(* Logix 5000 project; controller Universal_Device_Info_AOI_V0_1 vendor 1 type 14 code 176 rev 32.11; software revision 32.00; part 4 of 11 *)

           TBEN_L4_8IOL:O.Data[121].5   // IO-Link Port 8 - Output data word 7 (INT bit5)
           TBEN_L4_8IOL:O.Data[121].6   // IO-Link Port 8 - Output data word 7 (INT bit6)
           TBEN_L4_8IOL:O.Data[121].7   // IO-Link Port 8 - Output data word 7 (INT bit7)
           TBEN_L4_8IOL:O.Data[121].8   // IO-Link Port 8 - Output data word 7 (INT bit8)
           TBEN_L4_8IOL:O.Data[121].9   // IO-Link Port 8 - Output data word 7 (INT bit9)
           TBEN_L4_8IOL:O.Data[122]   // IO-Link Port 8 - Output data word 8
           TBEN_L4_8IOL:O.Data[122].0   // IO-Link Port 8 - Output data word 8 (INT bit0)
           TBEN_L4_8IOL:O.Data[122].1   // IO-Link Port 8 - Output data word 8 (INT bit1)
           TBEN_L4_8IOL:O.Data[122].10   // IO-Link Port 8 - Output data word 8 (INT bit10)
           TBEN_L4_8IOL:O.Data[122].11   // IO-Link Port 8 - Output data word 8 (INT bit11)
           TBEN_L4_8IOL:O.Data[122].12   // IO-Link Port 8 - Output data word 8 (INT bit12)
           TBEN_L4_8IOL:O.Data[122].13   // IO-Link Port 8 - Output data word 8 (INT bit13)
           TBEN_L4_8IOL:O.Data[122].14   // IO-Link Port 8 - Output data word 8 (INT bit14)
           TBEN_L4_8IOL:O.Data[122].15   // IO-Link Port 8 - Output data word 8 (INT bit15)
           TBEN_L4_8IOL:O.Data[122].2   // IO-Link Port 8 - Output data word 8 (INT bit2)
           TBEN_L4_8IOL:O.Data[122].3   // IO-Link Port 8 - Output data word 8 (INT bit3)
           TBEN_L4_8IOL:O.Data[122].4   // IO-Link Port 8 - Output data word 8 (INT bit4)
           TBEN_L4_8IOL:O.Data[122].5   // IO-Link Port 8 - Output data word 8 (INT bit5)
           TBEN_L4_8IOL:O.Data[122].6   // IO-Link Port 8 - Output data word 8 (INT bit6)
           TBEN_L4_8IOL:O.Data[122].7   // IO-Link Port 8 - Output data word 8 (INT bit7)
           TBEN_L4_8IOL:O.Data[122].8   // IO-Link Port 8 - Output data word 8 (INT bit8)
           TBEN_L4_8IOL:O.Data[122].9   // IO-Link Port 8 - Output data word 8 (INT bit9)
           TBEN_L4_8IOL:O.Data[123]   // IO-Link Port 8 - Output data word 9
           TBEN_L4_8IOL:O.Data[123].0   // IO-Link Port 8 - Output data word 9 (INT bit0)
           TBEN_L4_8IOL:O.Data[123].1   // IO-Link Port 8 - Output data word 9 (INT bit1)
           TBEN_L4_8IOL:O.Data[123].10   // IO-Link Port 8 - Output data word 9 (INT bit10)
           TBEN_L4_8IOL:O.Data[123].11   // IO-Link Port 8 - Output data word 9 (INT bit11)
           TBEN_L4_8IOL:O.Data[123].12   // IO-Link Port 8 - Output data word 9 (INT bit12)
           TBEN_L4_8IOL:O.Data[123].13   // IO-Link Port 8 - Output data word 9 (INT bit13)
           TBEN_L4_8IOL:O.Data[123].14   // IO-Link Port 8 - Output data word 9 (INT bit14)
           TBEN_L4_8IOL:O.Data[123].15   // IO-Link Port 8 - Output data word 9 (INT bit15)
           TBEN_L4_8IOL:O.Data[123].2   // IO-Link Port 8 - Output data word 9 (INT bit2)
           TBEN_L4_8IOL:O.Data[123].3   // IO-Link Port 8 - Output data word 9 (INT bit3)
           TBEN_L4_8IOL:O.Data[123].4   // IO-Link Port 8 - Output data word 9 (INT bit4)
           TBEN_L4_8IOL:O.Data[123].5   // IO-Link Port 8 - Output data word 9 (INT bit5)
           TBEN_L4_8IOL:O.Data[123].6   // IO-Link Port 8 - Output data word 9 (INT bit6)
           TBEN_L4_8IOL:O.Data[123].7   // IO-Link Port 8 - Output data word 9 (INT bit7)
           TBEN_L4_8IOL:O.Data[123].8   // IO-Link Port 8 - Output data word 9 (INT bit8)
           TBEN_L4_8IOL:O.Data[123].9   // IO-Link Port 8 - Output data word 9 (INT bit9)
           TBEN_L4_8IOL:O.Data[124]   // IO-Link Port 8 - Output data word 10
           TBEN_L4_8IOL:O.Data[124].0   // IO-Link Port 8 - Output data word 10 (INT bit0)
           TBEN_L4_8IOL:O.Data[124].1   // IO-Link Port 8 - Output data word 10 (INT bit1)
           TBEN_L4_8IOL:O.Data[124].10   // IO-Link Port 8 - Output data word 10 (INT bit10)
           TBEN_L4_8IOL:O.Data[124].11   // IO-Link Port 8 - Output data word 10 (INT bit11)
           TBEN_L4_8IOL:O.Data[124].12   // IO-Link Port 8 - Output data word 10 (INT bit12)
           TBEN_L4_8IOL:O.Data[124].13   // IO-Link Port 8 - Output data word 10 (INT bit13)
           TBEN_L4_8IOL:O.Data[124].14   // IO-Link Port 8 - Output data word 10 (INT bit14)
           TBEN_L4_8IOL:O.Data[124].15   // IO-Link Port 8 - Output data word 10 (INT bit15)
           TBEN_L4_8IOL:O.Data[124].2   // IO-Link Port 8 - Output data word 10 (INT bit2)
           TBEN_L4_8IOL:O.Data[124].3   // IO-Link Port 8 - Output data word 10 (INT bit3)
           TBEN_L4_8IOL:O.Data[124].4   // IO-Link Port 8 - Output data word 10 (INT bit4)
           TBEN_L4_8IOL:O.Data[124].5   // IO-Link Port 8 - Output data word 10 (INT bit5)
           TBEN_L4_8IOL:O.Data[124].6   // IO-Link Port 8 - Output data word 10 (INT bit6)
           TBEN_L4_8IOL:O.Data[124].7   // IO-Link Port 8 - Output data word 10 (INT bit7)
           TBEN_L4_8IOL:O.Data[124].8   // IO-Link Port 8 - Output data word 10 (INT bit8)
           TBEN_L4_8IOL:O.Data[124].9   // IO-Link Port 8 - Output data word 10 (INT bit9)
           TBEN_L4_8IOL:O.Data[125]   // IO-Link Port 8 - Output data word 11
           TBEN_L4_8IOL:O.Data[125].0   // IO-Link Port 8 - Output data word 11 (INT bit0)
           TBEN_L4_8IOL:O.Data[125].1   // IO-Link Port 8 - Output data word 11 (INT bit1)
           TBEN_L4_8IOL:O.Data[125].10   // IO-Link Port 8 - Output data word 11 (INT bit10)
           TBEN_L4_8IOL:O.Data[125].11   // IO-Link Port 8 - Output data word 11 (INT bit11)
           TBEN_L4_8IOL:O.Data[125].12   // IO-Link Port 8 - Output data word 11 (INT bit12)
           TBEN_L4_8IOL:O.Data[125].13   // IO-Link Port 8 - Output data word 11 (INT bit13)
           TBEN_L4_8IOL:O.Data[125].14   // IO-Link Port 8 - Output data word 11 (INT bit14)
           TBEN_L4_8IOL:O.Data[125].15   // IO-Link Port 8 - Output data word 11 (INT bit15)
           TBEN_L4_8IOL:O.Data[125].2   // IO-Link Port 8 - Output data word 11 (INT bit2)
           TBEN_L4_8IOL:O.Data[125].3   // IO-Link Port 8 - Output data word 11 (INT bit3)
           TBEN_L4_8IOL:O.Data[125].4   // IO-Link Port 8 - Output data word 11 (INT bit4)
           TBEN_L4_8IOL:O.Data[125].5   // IO-Link Port 8 - Output data word 11 (INT bit5)
           TBEN_L4_8IOL:O.Data[125].6   // IO-Link Port 8 - Output data word 11 (INT bit6)
           TBEN_L4_8IOL:O.Data[125].7   // IO-Link Port 8 - Output data word 11 (INT bit7)
           TBEN_L4_8IOL:O.Data[125].8   // IO-Link Port 8 - Output data word 11 (INT bit8)
           TBEN_L4_8IOL:O.Data[125].9   // IO-Link Port 8 - Output data word 11 (INT bit9)
           TBEN_L4_8IOL:O.Data[126]   // IO-Link Port 8 - Output data word 12
           TBEN_L4_8IOL:O.Data[126].0   // IO-Link Port 8 - Output data word 12 (INT bit0)
           TBEN_L4_8IOL:O.Data[126].1   // IO-Link Port 8 - Output data word 12 (INT bit1)
           TBEN_L4_8IOL:O.Data[126].10   // IO-Link Port 8 - Output data word 12 (INT bit10)
           TBEN_L4_8IOL:O.Data[126].11   // IO-Link Port 8 - Output data word 12 (INT bit11)
           TBEN_L4_8IOL:O.Data[126].12   // IO-Link Port 8 - Output data word 12 (INT bit12)
           TBEN_L4_8IOL:O.Data[126].13   // IO-Link Port 8 - Output data word 12 (INT bit13)
           TBEN_L4_8IOL:O.Data[126].14   // IO-Link Port 8 - Output data word 12 (INT bit14)
           TBEN_L4_8IOL:O.Data[126].15   // IO-Link Port 8 - Output data word 12 (INT bit15)
           TBEN_L4_8IOL:O.Data[126].2   // IO-Link Port 8 - Output data word 12 (INT bit2)
           TBEN_L4_8IOL:O.Data[126].3   // IO-Link Port 8 - Output data word 12 (INT bit3)
           TBEN_L4_8IOL:O.Data[126].4   // IO-Link Port 8 - Output data word 12 (INT bit4)
           TBEN_L4_8IOL:O.Data[126].5   // IO-Link Port 8 - Output data word 12 (INT bit5)
           TBEN_L4_8IOL:O.Data[126].6   // IO-Link Port 8 - Output data word 12 (INT bit6)
           TBEN_L4_8IOL:O.Data[126].7   // IO-Link Port 8 - Output data word 12 (INT bit7)
           TBEN_L4_8IOL:O.Data[126].8   // IO-Link Port 8 - Output data word 12 (INT bit8)
           TBEN_L4_8IOL:O.Data[126].9   // IO-Link Port 8 - Output data word 12 (INT bit9)
           TBEN_L4_8IOL:O.Data[127]   // IO-Link Port 8 - Output data word 13
           TBEN_L4_8IOL:O.Data[127].0   // IO-Link Port 8 - Output data word 13 (INT bit0)
           TBEN_L4_8IOL:O.Data[127].1   // IO-Link Port 8 - Output data word 13 (INT bit1)
           TBEN_L4_8IOL:O.Data[127].10   // IO-Link Port 8 - Output data word 13 (INT bit10)
           TBEN_L4_8IOL:O.Data[127].11   // IO-Link Port 8 - Output data word 13 (INT bit11)
           TBEN_L4_8IOL:O.Data[127].12   // IO-Link Port 8 - Output data word 13 (INT bit12)
           TBEN_L4_8IOL:O.Data[127].13   // IO-Link Port 8 - Output data word 13 (INT bit13)
           TBEN_L4_8IOL:O.Data[127].14   // IO-Link Port 8 - Output data word 13 (INT bit14)
           TBEN_L4_8IOL:O.Data[127].15   // IO-Link Port 8 - Output data word 13 (INT bit15)
           TBEN_L4_8IOL:O.Data[127].2   // IO-Link Port 8 - Output data word 13 (INT bit2)
           TBEN_L4_8IOL:O.Data[127].3   // IO-Link Port 8 - Output data word 13 (INT bit3)
           TBEN_L4_8IOL:O.Data[127].4   // IO-Link Port 8 - Output data word 13 (INT bit4)
           TBEN_L4_8IOL:O.Data[127].5   // IO-Link Port 8 - Output data word 13 (INT bit5)
           TBEN_L4_8IOL:O.Data[127].6   // IO-Link Port 8 - Output data word 13 (INT bit6)
           TBEN_L4_8IOL:O.Data[127].7   // IO-Link Port 8 - Output data word 13 (INT bit7)
           TBEN_L4_8IOL:O.Data[127].8   // IO-Link Port 8 - Output data word 13 (INT bit8)
           TBEN_L4_8IOL:O.Data[127].9   // IO-Link Port 8 - Output data word 13 (INT bit9)
           TBEN_L4_8IOL:O.Data[128]   // IO-Link Port 8 - Output data word 14
           TBEN_L4_8IOL:O.Data[128].0   // IO-Link Port 8 - Output data word 14 (INT bit0)
           TBEN_L4_8IOL:O.Data[128].1   // IO-Link Port 8 - Output data word 14 (INT bit1)
           TBEN_L4_8IOL:O.Data[128].10   // IO-Link Port 8 - Output data word 14 (INT bit10)
           TBEN_L4_8IOL:O.Data[128].11   // IO-Link Port 8 - Output data word 14 (INT bit11)
           TBEN_L4_8IOL:O.Data[128].12   // IO-Link Port 8 - Output data word 14 (INT bit12)
           TBEN_L4_8IOL:O.Data[128].13   // IO-Link Port 8 - Output data word 14 (INT bit13)
           TBEN_L4_8IOL:O.Data[128].14   // IO-Link Port 8 - Output data word 14 (INT bit14)
           TBEN_L4_8IOL:O.Data[128].15   // IO-Link Port 8 - Output data word 14 (INT bit15)
           TBEN_L4_8IOL:O.Data[128].2   // IO-Link Port 8 - Output data word 14 (INT bit2)
           TBEN_L4_8IOL:O.Data[128].3   // IO-Link Port 8 - Output data word 14 (INT bit3)
           TBEN_L4_8IOL:O.Data[128].4   // IO-Link Port 8 - Output data word 14 (INT bit4)
           TBEN_L4_8IOL:O.Data[128].5   // IO-Link Port 8 - Output data word 14 (INT bit5)
           TBEN_L4_8IOL:O.Data[128].6   // IO-Link Port 8 - Output data word 14 (INT bit6)
           TBEN_L4_8IOL:O.Data[128].7   // IO-Link Port 8 - Output data word 14 (INT bit7)
           TBEN_L4_8IOL:O.Data[128].8   // IO-Link Port 8 - Output data word 14 (INT bit8)
           TBEN_L4_8IOL:O.Data[128].9   // IO-Link Port 8 - Output data word 14 (INT bit9)
           TBEN_L4_8IOL:O.Data[129]   // IO-Link Port 8 - Output data word 15
           TBEN_L4_8IOL:O.Data[129].0   // IO-Link Port 8 - Output data word 15 (INT bit0)
           TBEN_L4_8IOL:O.Data[129].1   // IO-Link Port 8 - Output data word 15 (INT bit1)
           TBEN_L4_8IOL:O.Data[129].10   // IO-Link Port 8 - Output data word 15 (INT bit10)
           TBEN_L4_8IOL:O.Data[129].11   // IO-Link Port 8 - Output data word 15 (INT bit11)
           TBEN_L4_8IOL:O.Data[129].12   // IO-Link Port 8 - Output data word 15 (INT bit12)
           TBEN_L4_8IOL:O.Data[129].13   // IO-Link Port 8 - Output data word 15 (INT bit13)
           TBEN_L4_8IOL:O.Data[129].14   // IO-Link Port 8 - Output data word 15 (INT bit14)
           TBEN_L4_8IOL:O.Data[129].15   // IO-Link Port 8 - Output data word 15 (INT bit15)
           TBEN_L4_8IOL:O.Data[129].2   // IO-Link Port 8 - Output data word 15 (INT bit2)
           TBEN_L4_8IOL:O.Data[129].3   // IO-Link Port 8 - Output data word 15 (INT bit3)
           TBEN_L4_8IOL:O.Data[129].4   // IO-Link Port 8 - Output data word 15 (INT bit4)
           TBEN_L4_8IOL:O.Data[129].5   // IO-Link Port 8 - Output data word 15 (INT bit5)
           TBEN_L4_8IOL:O.Data[129].6   // IO-Link Port 8 - Output data word 15 (INT bit6)
           TBEN_L4_8IOL:O.Data[129].7   // IO-Link Port 8 - Output data word 15 (INT bit7)
           TBEN_L4_8IOL:O.Data[129].8   // IO-Link Port 8 - Output data word 15 (INT bit8)
           TBEN_L4_8IOL:O.Data[129].9   // IO-Link Port 8 - Output data word 15 (INT bit9)
           TBEN_L4_8IOL:O.Data[12]   // IO-Link Port 1 - Output data word 10
           TBEN_L4_8IOL:O.Data[12].0   // IO-Link Port 1 - Output data word 10 (INT bit0)
           TBEN_L4_8IOL:O.Data[12].1   // IO-Link Port 1 - Output data word 10 (INT bit1)
           TBEN_L4_8IOL:O.Data[12].10   // IO-Link Port 1 - Output data word 10 (INT bit10)
           TBEN_L4_8IOL:O.Data[12].11   // IO-Link Port 1 - Output data word 10 (INT bit11)
           TBEN_L4_8IOL:O.Data[12].12   // IO-Link Port 1 - Output data word 10 (INT bit12)
           TBEN_L4_8IOL:O.Data[12].13   // IO-Link Port 1 - Output data word 10 (INT bit13)
           TBEN_L4_8IOL:O.Data[12].14   // IO-Link Port 1 - Output data word 10 (INT bit14)
           TBEN_L4_8IOL:O.Data[12].15   // IO-Link Port 1 - Output data word 10 (INT bit15)
           TBEN_L4_8IOL:O.Data[12].2   // IO-Link Port 1 - Output data word 10 (INT bit2)
           TBEN_L4_8IOL:O.Data[12].3   // IO-Link Port 1 - Output data word 10 (INT bit3)
           TBEN_L4_8IOL:O.Data[12].4   // IO-Link Port 1 - Output data word 10 (INT bit4)
           TBEN_L4_8IOL:O.Data[12].5   // IO-Link Port 1 - Output data word 10 (INT bit5)
           TBEN_L4_8IOL:O.Data[12].6   // IO-Link Port 1 - Output data word 10 (INT bit6)
           TBEN_L4_8IOL:O.Data[12].7   // IO-Link Port 1 - Output data word 10 (INT bit7)
           TBEN_L4_8IOL:O.Data[12].8   // IO-Link Port 1 - Output data word 10 (INT bit8)
           TBEN_L4_8IOL:O.Data[12].9   // IO-Link Port 1 - Output data word 10 (INT bit9)
           TBEN_L4_8IOL:O.Data[130]   // VAUX1 Pin1 C0 (Ch0/1), VAUX1 Pin1 C1 (Ch2/3), VAUX1 Pin1 C2 (Ch4/5), VAUX1 Pin1 C3 (Ch6/7), VAUX1 Pin1 C4 (Ch8), VAUX1 Pin1 C5 (Ch10), VAUX1 Pin1 C6 (Ch12), VAUX1 Pin1 C7 (Ch14), VAUX2 Pin2 C4 (Ch9), VAUX2 Pin2 C5 (Ch11), VAUX2 Pin2 C6 (Ch13), VAUX2 Pin2 C7 (Ch15)
           TBEN_L4_8IOL:O.Data[130].0   // VAUX1 Pin1 C0 (Ch0/1) (ENUM bit0): 0=off, 1=on
           TBEN_L4_8IOL:O.Data[130].1   // VAUX1 Pin1 C1 (Ch2/3) (ENUM bit0): 0=off, 1=on
           TBEN_L4_8IOL:O.Data[130].10   // Reserved
           TBEN_L4_8IOL:O.Data[130].11   // Reserved
           TBEN_L4_8IOL:O.Data[130].12   // VAUX2 Pin2 C4 (Ch9) (ENUM bit0): 0=off, 1=on
           TBEN_L4_8IOL:O.Data[130].13   // VAUX2 Pin2 C5 (Ch11) (ENUM bit0): 0=off, 1=on
           TBEN_L4_8IOL:O.Data[130].14   // VAUX2 Pin2 C6 (Ch13) (ENUM bit0): 0=off, 1=on
           TBEN_L4_8IOL:O.Data[130].15   // VAUX2 Pin2 C7 (Ch15) (ENUM bit0): 0=off, 1=on
           TBEN_L4_8IOL:O.Data[130].2   // VAUX1 Pin1 C2 (Ch4/5) (ENUM bit0): 0=off, 1=on
           TBEN_L4_8IOL:O.Data[130].3   // VAUX1 Pin1 C3 (Ch6/7) (ENUM bit0): 0=off, 1=on
           TBEN_L4_8IOL:O.Data[130].4   // VAUX1 Pin1 C4 (Ch8) (ENUM bit0): 0=off, 1=on
           TBEN_L4_8IOL:O.Data[130].5   // VAUX1 Pin1 C5 (Ch10) (ENUM bit0): 0=off, 1=on
           TBEN_L4_8IOL:O.Data[130].6   // VAUX1 Pin1 C6 (Ch12) (ENUM bit0): 0=off, 1=on
           TBEN_L4_8IOL:O.Data[130].7   // VAUX1 Pin1 C7 (Ch14) (ENUM bit0): 0=off, 1=on
           TBEN_L4_8IOL:O.Data[130].8   // Reserved
           TBEN_L4_8IOL:O.Data[130].9   // Reserved
           TBEN_L4_8IOL:O.Data[13]   // IO-Link Port 1 - Output data word 11
           TBEN_L4_8IOL:O.Data[13].0   // IO-Link Port 1 - Output data word 11 (INT bit0)
           TBEN_L4_8IOL:O.Data[13].1   // IO-Link Port 1 - Output data word 11 (INT bit1)
           TBEN_L4_8IOL:O.Data[13].10   // IO-Link Port 1 - Output data word 11 (INT bit10)
           TBEN_L4_8IOL:O.Data[13].11   // IO-Link Port 1 - Output data word 11 (INT bit11)
           TBEN_L4_8IOL:O.Data[13].12   // IO-Link Port 1 - Output data word 11 (INT bit12)
           TBEN_L4_8IOL:O.Data[13].13   // IO-Link Port 1 - Output data word 11 (INT bit13)
           TBEN_L4_8IOL:O.Data[13].14   // IO-Link Port 1 - Output data word 11 (INT bit14)
           TBEN_L4_8IOL:O.Data[13].15   // IO-Link Port 1 - Output data word 11 (INT bit15)
           TBEN_L4_8IOL:O.Data[13].2   // IO-Link Port 1 - Output data word 11 (INT bit2)
           TBEN_L4_8IOL:O.Data[13].3   // IO-Link Port 1 - Output data word 11 (INT bit3)
           TBEN_L4_8IOL:O.Data[13].4   // IO-Link Port 1 - Output data word 11 (INT bit4)
           TBEN_L4_8IOL:O.Data[13].5   // IO-Link Port 1 - Output data word 11 (INT bit5)
           TBEN_L4_8IOL:O.Data[13].6   // IO-Link Port 1 - Output data word 11 (INT bit6)
           TBEN_L4_8IOL:O.Data[13].7   // IO-Link Port 1 - Output data word 11 (INT bit7)
           TBEN_L4_8IOL:O.Data[13].8   // IO-Link Port 1 - Output data word 11 (INT bit8)
           TBEN_L4_8IOL:O.Data[13].9   // IO-Link Port 1 - Output data word 11 (INT bit9)
           TBEN_L4_8IOL:O.Data[14]   // IO-Link Port 1 - Output data word 12
           TBEN_L4_8IOL:O.Data[14].0   // IO-Link Port 1 - Output data word 12 (INT bit0)
           TBEN_L4_8IOL:O.Data[14].1   // IO-Link Port 1 - Output data word 12 (INT bit1)
           TBEN_L4_8IOL:O.Data[14].10   // IO-Link Port 1 - Output data word 12 (INT bit10)
           TBEN_L4_8IOL:O.Data[14].11   // IO-Link Port 1 - Output data word 12 (INT bit11)
           TBEN_L4_8IOL:O.Data[14].12   // IO-Link Port 1 - Output data word 12 (INT bit12)
           TBEN_L4_8IOL:O.Data[14].13   // IO-Link Port 1 - Output data word 12 (INT bit13)
           TBEN_L4_8IOL:O.Data[14].14   // IO-Link Port 1 - Output data word 12 (INT bit14)
           TBEN_L4_8IOL:O.Data[14].15   // IO-Link Port 1 - Output data word 12 (INT bit15)
           TBEN_L4_8IOL:O.Data[14].2   // IO-Link Port 1 - Output data word 12 (INT bit2)
           TBEN_L4_8IOL:O.Data[14].3   // IO-Link Port 1 - Output data word 12 (INT bit3)
           TBEN_L4_8IOL:O.Data[14].4   // IO-Link Port 1 - Output data word 12 (INT bit4)
           TBEN_L4_8IOL:O.Data[14].5   // IO-Link Port 1 - Output data word 12 (INT bit5)
           TBEN_L4_8IOL:O.Data[14].6   // IO-Link Port 1 - Output data word 12 (INT bit6)
           TBEN_L4_8IOL:O.Data[14].7   // IO-Link Port 1 - Output data word 12 (INT bit7)
           TBEN_L4_8IOL:O.Data[14].8   // IO-Link Port 1 - Output data word 12 (INT bit8)
           TBEN_L4_8IOL:O.Data[14].9   // IO-Link Port 1 - Output data word 12 (INT bit9)
           TBEN_L4_8IOL:O.Data[15]   // IO-Link Port 1 - Output data word 13
           TBEN_L4_8IOL:O.Data[15].0   // IO-Link Port 1 - Output data word 13 (INT bit0)
           TBEN_L4_8IOL:O.Data[15].1   // IO-Link Port 1 - Output data word 13 (INT bit1)
           TBEN_L4_8IOL:O.Data[15].10   // IO-Link Port 1 - Output data word 13 (INT bit10)
           TBEN_L4_8IOL:O.Data[15].11   // IO-Link Port 1 - Output data word 13 (INT bit11)
           TBEN_L4_8IOL:O.Data[15].12   // IO-Link Port 1 - Output data word 13 (INT bit12)
           TBEN_L4_8IOL:O.Data[15].13   // IO-Link Port 1 - Output data word 13 (INT bit13)
           TBEN_L4_8IOL:O.Data[15].14   // IO-Link Port 1 - Output data word 13 (INT bit14)
           TBEN_L4_8IOL:O.Data[15].15   // IO-Link Port 1 - Output data word 13 (INT bit15)
           TBEN_L4_8IOL:O.Data[15].2   // IO-Link Port 1 - Output data word 13 (INT bit2)
           TBEN_L4_8IOL:O.Data[15].3   // IO-Link Port 1 - Output data word 13 (INT bit3)
           TBEN_L4_8IOL:O.Data[15].4   // IO-Link Port 1 - Output data word 13 (INT bit4)
           TBEN_L4_8IOL:O.Data[15].5   // IO-Link Port 1 - Output data word 13 (INT bit5)
           TBEN_L4_8IOL:O.Data[15].6   // IO-Link Port 1 - Output data word 13 (INT bit6)
           TBEN_L4_8IOL:O.Data[15].7   // IO-Link Port 1 - Output data word 13 (INT bit7)
           TBEN_L4_8IOL:O.Data[15].8   // IO-Link Port 1 - Output data word 13 (INT bit8)
           TBEN_L4_8IOL:O.Data[15].9   // IO-Link Port 1 - Output data word 13 (INT bit9)
           TBEN_L4_8IOL:O.Data[16]   // IO-Link Port 1 - Output data word 14
           TBEN_L4_8IOL:O.Data[16].0   // IO-Link Port 1 - Output data word 14 (INT bit0)
           TBEN_L4_8IOL:O.Data[16].1   // IO-Link Port 1 - Output data word 14 (INT bit1)
           TBEN_L4_8IOL:O.Data[16].10   // IO-Link Port 1 - Output data word 14 (INT bit10)
           TBEN_L4_8IOL:O.Data[16].11   // IO-Link Port 1 - Output data word 14 (INT bit11)
           TBEN_L4_8IOL:O.Data[16].12   // IO-Link Port 1 - Output data word 14 (INT bit12)
           TBEN_L4_8IOL:O.Data[16].13   // IO-Link Port 1 - Output data word 14 (INT bit13)
           TBEN_L4_8IOL:O.Data[16].14   // IO-Link Port 1 - Output data word 14 (INT bit14)
           TBEN_L4_8IOL:O.Data[16].15   // IO-Link Port 1 - Output data word 14 (INT bit15)
           TBEN_L4_8IOL:O.Data[16].2   // IO-Link Port 1 - Output data word 14 (INT bit2)
           TBEN_L4_8IOL:O.Data[16].3   // IO-Link Port 1 - Output data word 14 (INT bit3)
           TBEN_L4_8IOL:O.Data[16].4   // IO-Link Port 1 - Output data word 14 (INT bit4)
           TBEN_L4_8IOL:O.Data[16].5   // IO-Link Port 1 - Output data word 14 (INT bit5)
           TBEN_L4_8IOL:O.Data[16].6   // IO-Link Port 1 - Output data word 14 (INT bit6)
           TBEN_L4_8IOL:O.Data[16].7   // IO-Link Port 1 - Output data word 14 (INT bit7)
           TBEN_L4_8IOL:O.Data[16].8   // IO-Link Port 1 - Output data word 14 (INT bit8)
           TBEN_L4_8IOL:O.Data[16].9   // IO-Link Port 1 - Output data word 14 (INT bit9)
           TBEN_L4_8IOL:O.Data[17]   // IO-Link Port 1 - Output data word 15
           TBEN_L4_8IOL:O.Data[17].0   // IO-Link Port 1 - Output data word 15 (INT bit0)
           TBEN_L4_8IOL:O.Data[17].1   // IO-Link Port 1 - Output data word 15 (INT bit1)
           TBEN_L4_8IOL:O.Data[17].10   // IO-Link Port 1 - Output data word 15 (INT bit10)
           TBEN_L4_8IOL:O.Data[17].11   // IO-Link Port 1 - Output data word 15 (INT bit11)
           TBEN_L4_8IOL:O.Data[17].12   // IO-Link Port 1 - Output data word 15 (INT bit12)
           TBEN_L4_8IOL:O.Data[17].13   // IO-Link Port 1 - Output data word 15 (INT bit13)
           TBEN_L4_8IOL:O.Data[17].14   // IO-Link Port 1 - Output data word 15 (INT bit14)
           TBEN_L4_8IOL:O.Data[17].15   // IO-Link Port 1 - Output data word 15 (INT bit15)
           TBEN_L4_8IOL:O.Data[17].2   // IO-Link Port 1 - Output data word 15 (INT bit2)
           TBEN_L4_8IOL:O.Data[17].3   // IO-Link Port 1 - Output data word 15 (INT bit3)
           TBEN_L4_8IOL:O.Data[17].4   // IO-Link Port 1 - Output data word 15 (INT bit4)
           TBEN_L4_8IOL:O.Data[17].5   // IO-Link Port 1 - Output data word 15 (INT bit5)
           TBEN_L4_8IOL:O.Data[17].6   // IO-Link Port 1 - Output data word 15 (INT bit6)
           TBEN_L4_8IOL:O.Data[17].7   // IO-Link Port 1 - Output data word 15 (INT bit7)
           TBEN_L4_8IOL:O.Data[17].8   // IO-Link Port 1 - Output data word 15 (INT bit8)
           TBEN_L4_8IOL:O.Data[17].9   // IO-Link Port 1 - Output data word 15 (INT bit9)
           TBEN_L4_8IOL:O.Data[18]   // IO-Link Port 2 - Output data word 0
           TBEN_L4_8IOL:O.Data[18].0   // IO-Link Port 2 - Output data word 0 (INT bit0)
           TBEN_L4_8IOL:O.Data[18].1   // IO-Link Port 2 - Output data word 0 (INT bit1)
           TBEN_L4_8IOL:O.Data[18].10   // IO-Link Port 2 - Output data word 0 (INT bit10)
           TBEN_L4_8IOL:O.Data[18].11   // IO-Link Port 2 - Output data word 0 (INT bit11)
           TBEN_L4_8IOL:O.Data[18].12   // IO-Link Port 2 - Output data word 0 (INT bit12)
           TBEN_L4_8IOL:O.Data[18].13   // IO-Link Port 2 - Output data word 0 (INT bit13)
           TBEN_L4_8IOL:O.Data[18].14   // IO-Link Port 2 - Output data word 0 (INT bit14)
           TBEN_L4_8IOL:O.Data[18].15   // IO-Link Port 2 - Output data word 0 (INT bit15)
           TBEN_L4_8IOL:O.Data[18].2   // IO-Link Port 2 - Output data word 0 (INT bit2)
           TBEN_L4_8IOL:O.Data[18].3   // IO-Link Port 2 - Output data word 0 (INT bit3)
           TBEN_L4_8IOL:O.Data[18].4   // IO-Link Port 2 - Output data word 0 (INT bit4)
           TBEN_L4_8IOL:O.Data[18].5   // IO-Link Port 2 - Output data word 0 (INT bit5)
           TBEN_L4_8IOL:O.Data[18].6   // IO-Link Port 2 - Output data word 0 (INT bit6)
           TBEN_L4_8IOL:O.Data[18].7   // IO-Link Port 2 - Output data word 0 (INT bit7)
           TBEN_L4_8IOL:O.Data[18].8   // IO-Link Port 2 - Output data word 0 (INT bit8)
           TBEN_L4_8IOL:O.Data[18].9   // IO-Link Port 2 - Output data word 0 (INT bit9)
           TBEN_L4_8IOL:O.Data[19]   // IO-Link Port 2 - Output data word 1
           TBEN_L4_8IOL:O.Data[19].0   // IO-Link Port 2 - Output data word 1 (INT bit0)
           TBEN_L4_8IOL:O.Data[19].1   // IO-Link Port 2 - Output data word 1 (INT bit1)
           TBEN_L4_8IOL:O.Data[19].10   // IO-Link Port 2 - Output data word 1 (INT bit10)
           TBEN_L4_8IOL:O.Data[19].11   // IO-Link Port 2 - Output data word 1 (INT bit11)
           TBEN_L4_8IOL:O.Data[19].12   // IO-Link Port 2 - Output data word 1 (INT bit12)
           TBEN_L4_8IOL:O.Data[19].13   // IO-Link Port 2 - Output data word 1 (INT bit13)
           TBEN_L4_8IOL:O.Data[19].14   // IO-Link Port 2 - Output data word 1 (INT bit14)
           TBEN_L4_8IOL:O.Data[19].15   // IO-Link Port 2 - Output data word 1 (INT bit15)
           TBEN_L4_8IOL:O.Data[19].2   // IO-Link Port 2 - Output data word 1 (INT bit2)
           TBEN_L4_8IOL:O.Data[19].3   // IO-Link Port 2 - Output data word 1 (INT bit3)
           TBEN_L4_8IOL:O.Data[19].4   // IO-Link Port 2 - Output data word 1 (INT bit4)
           TBEN_L4_8IOL:O.Data[19].5   // IO-Link Port 2 - Output data word 1 (INT bit5)
           TBEN_L4_8IOL:O.Data[19].6   // IO-Link Port 2 - Output data word 1 (INT bit6)
           TBEN_L4_8IOL:O.Data[19].7   // IO-Link Port 2 - Output data word 1 (INT bit7)
           TBEN_L4_8IOL:O.Data[19].8   // IO-Link Port 2 - Output data word 1 (INT bit8)
           TBEN_L4_8IOL:O.Data[19].9   // IO-Link Port 2 - Output data word 1 (INT bit9)
           TBEN_L4_8IOL:O.Data[1]   // DXP 1 - DXP Output value, DXP 3 - DXP Output value, DXP 5 - DXP Output value, DXP 7 - DXP Output value
           TBEN_L4_8IOL:O.Data[1].0   // Reserved
           TBEN_L4_8IOL:O.Data[1].1   // DXP 1 - DXP Output value (ENUM bit0): 0=off, 1=on
           TBEN_L4_8IOL:O.Data[1].10   // Reserved
           TBEN_L4_8IOL:O.Data[1].11   // Reserved
           TBEN_L4_8IOL:O.Data[1].12   // Reserved
           TBEN_L4_8IOL:O.Data[1].13   // Reserved
           TBEN_L4_8IOL:O.Data[1].14   // Reserved
           TBEN_L4_8IOL:O.Data[1].15   // Reserved
           TBEN_L4_8IOL:O.Data[1].2   // Reserved
           TBEN_L4_8IOL:O.Data[1].3   // DXP 3 - DXP Output value (ENUM bit0): 0=off, 1=on
           TBEN_L4_8IOL:O.Data[1].4   // Reserved
           TBEN_L4_8IOL:O.Data[1].5   // DXP 5 - DXP Output value (ENUM bit0): 0=off, 1=on
           TBEN_L4_8IOL:O.Data[1].6   // Reserved
           TBEN_L4_8IOL:O.Data[1].7   // DXP 7 - DXP Output value (ENUM bit0): 0=off, 1=on
           TBEN_L4_8IOL:O.Data[1].8   // Reserved
           TBEN_L4_8IOL:O.Data[1].9   // Reserved
           TBEN_L4_8IOL:O.Data[20]   // IO-Link Port 2 - Output data word 2
           TBEN_L4_8IOL:O.Data[20].0   // IO-Link Port 2 - Output data word 2 (INT bit0)
           TBEN_L4_8IOL:O.Data[20].1   // IO-Link Port 2 - Output data word 2 (INT bit1)
           TBEN_L4_8IOL:O.Data[20].10   // IO-Link Port 2 - Output data word 2 (INT bit10)
           TBEN_L4_8IOL:O.Data[20].11   // IO-Link Port 2 - Output data word 2 (INT bit11)
           TBEN_L4_8IOL:O.Data[20].12   // IO-Link Port 2 - Output data word 2 (INT bit12)
           TBEN_L4_8IOL:O.Data[20].13   // IO-Link Port 2 - Output data word 2 (INT bit13)
           TBEN_L4_8IOL:O.Data[20].14   // IO-Link Port 2 - Output data word 2 (INT bit14)
           TBEN_L4_8IOL:O.Data[20].15   // IO-Link Port 2 - Output data word 2 (INT bit15)
           TBEN_L4_8IOL:O.Data[20].2   // IO-Link Port 2 - Output data word 2 (INT bit2)
           TBEN_L4_8IOL:O.Data[20].3   // IO-Link Port 2 - Output data word 2 (INT bit3)
           TBEN_L4_8IOL:O.Data[20].4   // IO-Link Port 2 - Output data word 2 (INT bit4)
           TBEN_L4_8IOL:O.Data[20].5   // IO-Link Port 2 - Output data word 2 (INT bit5)
           TBEN_L4_8IOL:O.Data[20].6   // IO-Link Port 2 - Output data word 2 (INT bit6)
           TBEN_L4_8IOL:O.Data[20].7   // IO-Link Port 2 - Output data word 2 (INT bit7)
           TBEN_L4_8IOL:O.Data[20].8   // IO-Link Port 2 - Output data word 2 (INT bit8)
           TBEN_L4_8IOL:O.Data[20].9   // IO-Link Port 2 - Output data word 2 (INT bit9)
           TBEN_L4_8IOL:O.Data[21]   // IO-Link Port 2 - Output data word 3
           TBEN_L4_8IOL:O.Data[21].0   // IO-Link Port 2 - Output data word 3 (INT bit0)
           TBEN_L4_8IOL:O.Data[21].1   // IO-Link Port 2 - Output data word 3 (INT bit1)
           TBEN_L4_8IOL:O.Data[21].10   // IO-Link Port 2 - Output data word 3 (INT bit10)
           TBEN_L4_8IOL:O.Data[21].11   // IO-Link Port 2 - Output data word 3 (INT bit11)
           TBEN_L4_8IOL:O.Data[21].12   // IO-Link Port 2 - Output data word 3 (INT bit12)
           TBEN_L4_8IOL:O.Data[21].13   // IO-Link Port 2 - Output data word 3 (INT bit13)
           TBEN_L4_8IOL:O.Data[21].14   // IO-Link Port 2 - Output data word 3 (INT bit14)
           TBEN_L4_8IOL:O.Data[21].15   // IO-Link Port 2 - Output data word 3 (INT bit15)
           TBEN_L4_8IOL:O.Data[21].2   // IO-Link Port 2 - Output data word 3 (INT bit2)
           TBEN_L4_8IOL:O.Data[21].3   // IO-Link Port 2 - Output data word 3 (INT bit3)
           TBEN_L4_8IOL:O.Data[21].4   // IO-Link Port 2 - Output data word 3 (INT bit4)
           TBEN_L4_8IOL:O.Data[21].5   // IO-Link Port 2 - Output data word 3 (INT bit5)
           TBEN_L4_8IOL:O.Data[21].6   // IO-Link Port 2 - Output data word 3 (INT bit6)
           TBEN_L4_8IOL:O.Data[21].7   // IO-Link Port 2 - Output data word 3 (INT bit7)
           TBEN_L4_8IOL:O.Data[21].8   // IO-Link Port 2 - Output data word 3 (INT bit8)
           TBEN_L4_8IOL:O.Data[21].9   // IO-Link Port 2 - Output data word 3 (INT bit9)
           TBEN_L4_8IOL:O.Data[22]   // IO-Link Port 2 - Output data word 4
           TBEN_L4_8IOL:O.Data[22].0   // IO-Link Port 2 - Output data word 4 (INT bit0)
           TBEN_L4_8IOL:O.Data[22].1   // IO-Link Port 2 - Output data word 4 (INT bit1)
           TBEN_L4_8IOL:O.Data[22].10   // IO-Link Port 2 - Output data word 4 (INT bit10)
           TBEN_L4_8IOL:O.Data[22].11   // IO-Link Port 2 - Output data word 4 (INT bit11)
           TBEN_L4_8IOL:O.Data[22].12   // IO-Link Port 2 - Output data word 4 (INT bit12)
           TBEN_L4_8IOL:O.Data[22].13   // IO-Link Port 2 - Output data word 4 (INT bit13)
           TBEN_L4_8IOL:O.Data[22].14   // IO-Link Port 2 - Output data word 4 (INT bit14)
           TBEN_L4_8IOL:O.Data[22].15   // IO-Link Port 2 - Output data word 4 (INT bit15)
           TBEN_L4_8IOL:O.Data[22].2   // IO-Link Port 2 - Output data word 4 (INT bit2)
           TBEN_L4_8IOL:O.Data[22].3   // IO-Link Port 2 - Output data word 4 (INT bit3)
           TBEN_L4_8IOL:O.Data[22].4   // IO-Link Port 2 - Output data word 4 (INT bit4)
           TBEN_L4_8IOL:O.Data[22].5   // IO-Link Port 2 - Output data word 4 (INT bit5)
           TBEN_L4_8IOL:O.Data[22].6   // IO-Link Port 2 - Output data word 4 (INT bit6)
           TBEN_L4_8IOL:O.Data[22].7   // IO-Link Port 2 - Output data word 4 (INT bit7)
           TBEN_L4_8IOL:O.Data[22].8   // IO-Link Port 2 - Output data word 4 (INT bit8)
           TBEN_L4_8IOL:O.Data[22].9   // IO-Link Port 2 - Output data word 4 (INT bit9)
           TBEN_L4_8IOL:O.Data[23]   // IO-Link Port 2 - Output data word 5
           TBEN_L4_8IOL:O.Data[23].0   // IO-Link Port 2 - Output data word 5 (INT bit0)
           TBEN_L4_8IOL:O.Data[23].1   // IO-Link Port 2 - Output data word 5 (INT bit1)
           TBEN_L4_8IOL:O.Data[23].10   // IO-Link Port 2 - Output data word 5 (INT bit10)
           TBEN_L4_8IOL:O.Data[23].11   // IO-Link Port 2 - Output data word 5 (INT bit11)
           TBEN_L4_8IOL:O.Data[23].12   // IO-Link Port 2 - Output data word 5 (INT bit12)
           TBEN_L4_8IOL:O.Data[23].13   // IO-Link Port 2 - Output data word 5 (INT bit13)
           TBEN_L4_8IOL:O.Data[23].14   // IO-Link Port 2 - Output data word 5 (INT bit14)
           TBEN_L4_8IOL:O.Data[23].15   // IO-Link Port 2 - Output data word 5 (INT bit15)
           TBEN_L4_8IOL:O.Data[23].2   // IO-Link Port 2 - Output data word 5 (INT bit2)
           TBEN_L4_8IOL:O.Data[23].3   // IO-Link Port 2 - Output data word 5 (INT bit3)
           TBEN_L4_8IOL:O.Data[23].4   // IO-Link Port 2 - Output data word 5 (INT bit4)
           TBEN_L4_8IOL:O.Data[23].5   // IO-Link Port 2 - Output data word 5 (INT bit5)
           TBEN_L4_8IOL:O.Data[23].6   // IO-Link Port 2 - Output data word 5 (INT bit6)
           TBEN_L4_8IOL:O.Data[23].7   // IO-Link Port 2 - Output data word 5 (INT bit7)
           TBEN_L4_8IOL:O.Data[23].8   // IO-Link Port 2 - Output data word 5 (INT bit8)
           TBEN_L4_8IOL:O.Data[23].9   // IO-Link Port 2 - Output data word 5 (INT bit9)
           TBEN_L4_8IOL:O.Data[24]   // IO-Link Port 2 - Output data word 6
           TBEN_L4_8IOL:O.Data[24].0   // IO-Link Port 2 - Output data word 6 (INT bit0)
           TBEN_L4_8IOL:O.Data[24].1   // IO-Link Port 2 - Output data word 6 (INT bit1)
           TBEN_L4_8IOL:O.Data[24].10   // IO-Link Port 2 - Output data word 6 (INT bit10)
           TBEN_L4_8IOL:O.Data[24].11   // IO-Link Port 2 - Output data word 6 (INT bit11)
           TBEN_L4_8IOL:O.Data[24].12   // IO-Link Port 2 - Output data word 6 (INT bit12)
           TBEN_L4_8IOL:O.Data[24].13   // IO-Link Port 2 - Output data word 6 (INT bit13)
           TBEN_L4_8IOL:O.Data[24].14   // IO-Link Port 2 - Output data word 6 (INT bit14)
           TBEN_L4_8IOL:O.Data[24].15   // IO-Link Port 2 - Output data word 6 (INT bit15)
           TBEN_L4_8IOL:O.Data[24].2   // IO-Link Port 2 - Output data word 6 (INT bit2)
           TBEN_L4_8IOL:O.Data[24].3   // IO-Link Port 2 - Output data word 6 (INT bit3)
           TBEN_L4_8IOL:O.Data[24].4   // IO-Link Port 2 - Output data word 6 (INT bit4)
           TBEN_L4_8IOL:O.Data[24].5   // IO-Link Port 2 - Output data word 6 (INT bit5)
           TBEN_L4_8IOL:O.Data[24].6   // IO-Link Port 2 - Output data word 6 (INT bit6)
           TBEN_L4_8IOL:O.Data[24].7   // IO-Link Port 2 - Output data word 6 (INT bit7)
           TBEN_L4_8IOL:O.Data[24].8   // IO-Link Port 2 - Output data word 6 (INT bit8)
           TBEN_L4_8IOL:O.Data[24].9   // IO-Link Port 2 - Output data word 6 (INT bit9)
           TBEN_L4_8IOL:O.Data[25]   // IO-Link Port 2 - Output data word 7
           TBEN_L4_8IOL:O.Data[25].0   // IO-Link Port 2 - Output data word 7 (INT bit0)
           TBEN_L4_8IOL:O.Data[25].1   // IO-Link Port 2 - Output data word 7 (INT bit1)
           TBEN_L4_8IOL:O.Data[25].10   // IO-Link Port 2 - Output data word 7 (INT bit10)
           TBEN_L4_8IOL:O.Data[25].11   // IO-Link Port 2 - Output data word 7 (INT bit11)
           TBEN_L4_8IOL:O.Data[25].12   // IO-Link Port 2 - Output data word 7 (INT bit12)
           TBEN_L4_8IOL:O.Data[25].13   // IO-Link Port 2 - Output data word 7 (INT bit13)
           TBEN_L4_8IOL:O.Data[25].14   // IO-Link Port 2 - Output data word 7 (INT bit14)
           TBEN_L4_8IOL:O.Data[25].15   // IO-Link Port 2 - Output data word 7 (INT bit15)
           TBEN_L4_8IOL:O.Data[25].2   // IO-Link Port 2 - Output data word 7 (INT bit2)
           TBEN_L4_8IOL:O.Data[25].3   // IO-Link Port 2 - Output data word 7 (INT bit3)
           TBEN_L4_8IOL:O.Data[25].4   // IO-Link Port 2 - Output data word 7 (INT bit4)
           TBEN_L4_8IOL:O.Data[25].5   // IO-Link Port 2 - Output data word 7 (INT bit5)
           TBEN_L4_8IOL:O.Data[25].6   // IO-Link Port 2 - Output data word 7 (INT bit6)
           TBEN_L4_8IOL:O.Data[25].7   // IO-Link Port 2 - Output data word 7 (INT bit7)
           TBEN_L4_8IOL:O.Data[25].8   // IO-Link Port 2 - Output data word 7 (INT bit8)
           TBEN_L4_8IOL:O.Data[25].9   // IO-Link Port 2 - Output data word 7 (INT bit9)
           TBEN_L4_8IOL:O.Data[26]   // IO-Link Port 2 - Output data word 8
           TBEN_L4_8IOL:O.Data[26].0   // IO-Link Port 2 - Output data word 8 (INT bit0)
           TBEN_L4_8IOL:O.Data[26].1   // IO-Link Port 2 - Output data word 8 (INT bit1)
           TBEN_L4_8IOL:O.Data[26].10   // IO-Link Port 2 - Output data word 8 (INT bit10)
           TBEN_L4_8IOL:O.Data[26].11   // IO-Link Port 2 - Output data word 8 (INT bit11)
           TBEN_L4_8IOL:O.Data[26].12   // IO-Link Port 2 - Output data word 8 (INT bit12)
           TBEN_L4_8IOL:O.Data[26].13   // IO-Link Port 2 - Output data word 8 (INT bit13)
           TBEN_L4_8IOL:O.Data[26].14   // IO-Link Port 2 - Output data word 8 (INT bit14)
           TBEN_L4_8IOL:O.Data[26].15   // IO-Link Port 2 - Output data word 8 (INT bit15)
           TBEN_L4_8IOL:O.Data[26].2   // IO-Link Port 2 - Output data word 8 (INT bit2)
           TBEN_L4_8IOL:O.Data[26].3   // IO-Link Port 2 - Output data word 8 (INT bit3)
           TBEN_L4_8IOL:O.Data[26].4   // IO-Link Port 2 - Output data word 8 (INT bit4)
           TBEN_L4_8IOL:O.Data[26].5   // IO-Link Port 2 - Output data word 8 (INT bit5)
           TBEN_L4_8IOL:O.Data[26].6   // IO-Link Port 2 - Output data word 8 (INT bit6)
           TBEN_L4_8IOL:O.Data[26].7   // IO-Link Port 2 - Output data word 8 (INT bit7)
           TBEN_L4_8IOL:O.Data[26].8   // IO-Link Port 2 - Output data word 8 (INT bit8)
           TBEN_L4_8IOL:O.Data[26].9   // IO-Link Port 2 - Output data word 8 (INT bit9)
           TBEN_L4_8IOL:O.Data[27]   // IO-Link Port 2 - Output data word 9
           TBEN_L4_8IOL:O.Data[27].0   // IO-Link Port 2 - Output data word 9 (INT bit0)
           TBEN_L4_8IOL:O.Data[27].1   // IO-Link Port 2 - Output data word 9 (INT bit1)
           TBEN_L4_8IOL:O.Data[27].10   // IO-Link Port 2 - Output data word 9 (INT bit10)
           TBEN_L4_8IOL:O.Data[27].11   // IO-Link Port 2 - Output data word 9 (INT bit11)
           TBEN_L4_8IOL:O.Data[27].12   // IO-Link Port 2 - Output data word 9 (INT bit12)
           TBEN_L4_8IOL:O.Data[27].13   // IO-Link Port 2 - Output data word 9 (INT bit13)
           TBEN_L4_8IOL:O.Data[27].14   // IO-Link Port 2 - Output data word 9 (INT bit14)
           TBEN_L4_8IOL:O.Data[27].15   // IO-Link Port 2 - Output data word 9 (INT bit15)
           TBEN_L4_8IOL:O.Data[27].2   // IO-Link Port 2 - Output data word 9 (INT bit2)
           TBEN_L4_8IOL:O.Data[27].3   // IO-Link Port 2 - Output data word 9 (INT bit3)
           TBEN_L4_8IOL:O.Data[27].4   // IO-Link Port 2 - Output data word 9 (INT bit4)
           TBEN_L4_8IOL:O.Data[27].5   // IO-Link Port 2 - Output data word 9 (INT bit5)
           TBEN_L4_8IOL:O.Data[27].6   // IO-Link Port 2 - Output data word 9 (INT bit6)
           TBEN_L4_8IOL:O.Data[27].7   // IO-Link Port 2 - Output data word 9 (INT bit7)
           TBEN_L4_8IOL:O.Data[27].8   // IO-Link Port 2 - Output data word 9 (INT bit8)
           TBEN_L4_8IOL:O.Data[27].9   // IO-Link Port 2 - Output data word 9 (INT bit9)
           TBEN_L4_8IOL:O.Data[28]   // IO-Link Port 2 - Output data word 10
           TBEN_L4_8IOL:O.Data[28].0   // IO-Link Port 2 - Output data word 10 (INT bit0)
           TBEN_L4_8IOL:O.Data[28].1   // IO-Link Port 2 - Output data word 10 (INT bit1)
           TBEN_L4_8IOL:O.Data[28].10   // IO-Link Port 2 - Output data word 10 (INT bit10)
           TBEN_L4_8IOL:O.Data[28].11   // IO-Link Port 2 - Output data word 10 (INT bit11)
           TBEN_L4_8IOL:O.Data[28].12   // IO-Link Port 2 - Output data word 10 (INT bit12)
           TBEN_L4_8IOL:O.Data[28].13   // IO-Link Port 2 - Output data word 10 (INT bit13)
           TBEN_L4_8IOL:O.Data[28].14   // IO-Link Port 2 - Output data word 10 (INT bit14)
           TBEN_L4_8IOL:O.Data[28].15   // IO-Link Port 2 - Output data word 10 (INT bit15)
           TBEN_L4_8IOL:O.Data[28].2   // IO-Link Port 2 - Output data word 10 (INT bit2)
           TBEN_L4_8IOL:O.Data[28].3   // IO-Link Port 2 - Output data word 10 (INT bit3)
           TBEN_L4_8IOL:O.Data[28].4   // IO-Link Port 2 - Output data word 10 (INT bit4)
           TBEN_L4_8IOL:O.Data[28].5   // IO-Link Port 2 - Output data word 10 (INT bit5)
           TBEN_L4_8IOL:O.Data[28].6   // IO-Link Port 2 - Output data word 10 (INT bit6)
           TBEN_L4_8IOL:O.Data[28].7   // IO-Link Port 2 - Output data word 10 (INT bit7)
           TBEN_L4_8IOL:O.Data[28].8   // IO-Link Port 2 - Output data word 10 (INT bit8)
           TBEN_L4_8IOL:O.Data[28].9   // IO-Link Port 2 - Output data word 10 (INT bit9)
           TBEN_L4_8IOL:O.Data[29]   // IO-Link Port 2 - Output data word 11
           TBEN_L4_8IOL:O.Data[29].0   // IO-Link Port 2 - Output data word 11 (INT bit0)
           TBEN_L4_8IOL:O.Data[29].1   // IO-Link Port 2 - Output data word 11 (INT bit1)
           TBEN_L4_8IOL:O.Data[29].10   // IO-Link Port 2 - Output data word 11 (INT bit10)
           TBEN_L4_8IOL:O.Data[29].11   // IO-Link Port 2 - Output data word 11 (INT bit11)
           TBEN_L4_8IOL:O.Data[29].12   // IO-Link Port 2 - Output data word 11 (INT bit12)
           TBEN_L4_8IOL:O.Data[29].13   // IO-Link Port 2 - Output data word 11 (INT bit13)
           TBEN_L4_8IOL:O.Data[29].14   // IO-Link Port 2 - Output data word 11 (INT bit14)
           TBEN_L4_8IOL:O.Data[29].15   // IO-Link Port 2 - Output data word 11 (INT bit15)
           TBEN_L4_8IOL:O.Data[29].2   // IO-Link Port 2 - Output data word 11 (INT bit2)
           TBEN_L4_8IOL:O.Data[29].3   // IO-Link Port 2 - Output data word 11 (INT bit3)
           TBEN_L4_8IOL:O.Data[29].4   // IO-Link Port 2 - Output data word 11 (INT bit4)
           TBEN_L4_8IOL:O.Data[29].5   // IO-Link Port 2 - Output data word 11 (INT bit5)
           TBEN_L4_8IOL:O.Data[29].6   // IO-Link Port 2 - Output data word 11 (INT bit6)
           TBEN_L4_8IOL:O.Data[29].7   // IO-Link Port 2 - Output data word 11 (INT bit7)
           TBEN_L4_8IOL:O.Data[29].8   // IO-Link Port 2 - Output data word 11 (INT bit8)
           TBEN_L4_8IOL:O.Data[29].9   // IO-Link Port 2 - Output data word 11 (INT bit9)
           TBEN_L4_8IOL:O.Data[2]   // IO-Link Port 1 - Output data word 0
           TBEN_L4_8IOL:O.Data[2].0   // IO-Link Port 1 - Output data word 0 (INT bit0)
           TBEN_L4_8IOL:O.Data[2].1   // IO-Link Port 1 - Output data word 0 (INT bit1)
           TBEN_L4_8IOL:O.Data[2].10   // IO-Link Port 1 - Output data word 0 (INT bit10)
           TBEN_L4_8IOL:O.Data[2].11   // IO-Link Port 1 - Output data word 0 (INT bit11)
           TBEN_L4_8IOL:O.Data[2].12   // IO-Link Port 1 - Output data word 0 (INT bit12)
           TBEN_L4_8IOL:O.Data[2].13   // IO-Link Port 1 - Output data word 0 (INT bit13)
           TBEN_L4_8IOL:O.Data[2].14   // IO-Link Port 1 - Output data word 0 (INT bit14)
           TBEN_L4_8IOL:O.Data[2].15   // IO-Link Port 1 - Output data word 0 (INT bit15)
           TBEN_L4_8IOL:O.Data[2].2   // IO-Link Port 1 - Output data word 0 (INT bit2)
           TBEN_L4_8IOL:O.Data[2].3   // IO-Link Port 1 - Output data word 0 (INT bit3)
           TBEN_L4_8IOL:O.Data[2].4   // IO-Link Port 1 - Output data word 0 (INT bit4)
           TBEN_L4_8IOL:O.Data[2].5   // IO-Link Port 1 - Output data word 0 (INT bit5)
           TBEN_L4_8IOL:O.Data[2].6   // IO-Link Port 1 - Output data word 0 (INT bit6)
           TBEN_L4_8IOL:O.Data[2].7   // IO-Link Port 1 - Output data word 0 (INT bit7)
           TBEN_L4_8IOL:O.Data[2].8   // IO-Link Port 1 - Output data word 0 (INT bit8)
           TBEN_L4_8IOL:O.Data[2].9   // IO-Link Port 1 - Output data word 0 (INT bit9)
           TBEN_L4_8IOL:O.Data[30]   // IO-Link Port 2 - Output data word 12
           TBEN_L4_8IOL:O.Data[30].0   // IO-Link Port 2 - Output data word 12 (INT bit0)
           TBEN_L4_8IOL:O.Data[30].1   // IO-Link Port 2 - Output data word 12 (INT bit1)
           TBEN_L4_8IOL:O.Data[30].10   // IO-Link Port 2 - Output data word 12 (INT bit10)
           TBEN_L4_8IOL:O.Data[30].11   // IO-Link Port 2 - Output data word 12 (INT bit11)
           TBEN_L4_8IOL:O.Data[30].12   // IO-Link Port 2 - Output data word 12 (INT bit12)
           TBEN_L4_8IOL:O.Data[30].13   // IO-Link Port 2 - Output data word 12 (INT bit13)
           TBEN_L4_8IOL:O.Data[30].14   // IO-Link Port 2 - Output data word 12 (INT bit14)
           TBEN_L4_8IOL:O.Data[30].15   // IO-Link Port 2 - Output data word 12 (INT bit15)
           TBEN_L4_8IOL:O.Data[30].2   // IO-Link Port 2 - Output data word 12 (INT bit2)
           TBEN_L4_8IOL:O.Data[30].3   // IO-Link Port 2 - Output data word 12 (INT bit3)
           TBEN_L4_8IOL:O.Data[30].4   // IO-Link Port 2 - Output data word 12 (INT bit4)
           TBEN_L4_8IOL:O.Data[30].5   // IO-Link Port 2 - Output data word 12 (INT bit5)
           TBEN_L4_8IOL:O.Data[30].6   // IO-Link Port 2 - Output data word 12 (INT bit6)
           TBEN_L4_8IOL:O.Data[30].7   // IO-Link Port 2 - Output data word 12 (INT bit7)
           TBEN_L4_8IOL:O.Data[30].8   // IO-Link Port 2 - Output data word 12 (INT bit8)
           TBEN_L4_8IOL:O.Data[30].9   // IO-Link Port 2 - Output data word 12 (INT bit9)
           TBEN_L4_8IOL:O.Data[31]   // IO-Link Port 2 - Output data word 13
           TBEN_L4_8IOL:O.Data[31].0   // IO-Link Port 2 - Output data word 13 (INT bit0)
           TBEN_L4_8IOL:O.Data[31].1   // IO-Link Port 2 - Output data word 13 (INT bit1)
           TBEN_L4_8IOL:O.Data[31].10   // IO-Link Port 2 - Output data word 13 (INT bit10)
           TBEN_L4_8IOL:O.Data[31].11   // IO-Link Port 2 - Output data word 13 (INT bit11)
           TBEN_L4_8IOL:O.Data[31].12   // IO-Link Port 2 - Output data word 13 (INT bit12)
           TBEN_L4_8IOL:O.Data[31].13   // IO-Link Port 2 - Output data word 13 (INT bit13)
           TBEN_L4_8IOL:O.Data[31].14   // IO-Link Port 2 - Output data word 13 (INT bit14)
           TBEN_L4_8IOL:O.Data[31].15   // IO-Link Port 2 - Output data word 13 (INT bit15)
           TBEN_L4_8IOL:O.Data[31].2   // IO-Link Port 2 - Output data word 13 (INT bit2)
           TBEN_L4_8IOL:O.Data[31].3   // IO-Link Port 2 - Output data word 13 (INT bit3)
           TBEN_L4_8IOL:O.Data[31].4   // IO-Link Port 2 - Output data word 13 (INT bit4)
           TBEN_L4_8IOL:O.Data[31].5   // IO-Link Port 2 - Output data word 13 (INT bit5)
           TBEN_L4_8IOL:O.Data[31].6   // IO-Link Port 2 - Output data word 13 (INT bit6)
           TBEN_L4_8IOL:O.Data[31].7   // IO-Link Port 2 - Output data word 13 (INT bit7)
           TBEN_L4_8IOL:O.Data[31].8   // IO-Link Port 2 - Output data word 13 (INT bit8)
           TBEN_L4_8IOL:O.Data[31].9   // IO-Link Port 2 - Output data word 13 (INT bit9)
           TBEN_L4_8IOL:O.Data[32]   // IO-Link Port 2 - Output data word 14
           TBEN_L4_8IOL:O.Data[32].0   // IO-Link Port 2 - Output data word 14 (INT bit0)
           TBEN_L4_8IOL:O.Data[32].1   // IO-Link Port 2 - Output data word 14 (INT bit1)
           TBEN_L4_8IOL:O.Data[32].10   // IO-Link Port 2 - Output data word 14 (INT bit10)
           TBEN_L4_8IOL:O.Data[32].11   // IO-Link Port 2 - Output data word 14 (INT bit11)
           TBEN_L4_8IOL:O.Data[32].12   // IO-Link Port 2 - Output data word 14 (INT bit12)
           TBEN_L4_8IOL:O.Data[32].13   // IO-Link Port 2 - Output data word 14 (INT bit13)
           TBEN_L4_8IOL:O.Data[32].14   // IO-Link Port 2 - Output data word 14 (INT bit14)
           TBEN_L4_8IOL:O.Data[32].15   // IO-Link Port 2 - Output data word 14 (INT bit15)
           TBEN_L4_8IOL:O.Data[32].2   // IO-Link Port 2 - Output data word 14 (INT bit2)
           TBEN_L4_8IOL:O.Data[32].3   // IO-Link Port 2 - Output data word 14 (INT bit3)
           TBEN_L4_8IOL:O.Data[32].4   // IO-Link Port 2 - Output data word 14 (INT bit4)
           TBEN_L4_8IOL:O.Data[32].5   // IO-Link Port 2 - Output data word 14 (INT bit5)
           TBEN_L4_8IOL:O.Data[32].6   // IO-Link Port 2 - Output data word 14 (INT bit6)
           TBEN_L4_8IOL:O.Data[32].7   // IO-Link Port 2 - Output data word 14 (INT bit7)
           TBEN_L4_8IOL:O.Data[32].8   // IO-Link Port 2 - Output data word 14 (INT bit8)
           TBEN_L4_8IOL:O.Data[32].9   // IO-Link Port 2 - Output data word 14 (INT bit9)
           TBEN_L4_8IOL:O.Data[33]   // IO-Link Port 2 - Output data word 15
           TBEN_L4_8IOL:O.Data[33].0   // IO-Link Port 2 - Output data word 15 (INT bit0)
           TBEN_L4_8IOL:O.Data[33].1   // IO-Link Port 2 - Output data word 15 (INT bit1)
           TBEN_L4_8IOL:O.Data[33].10   // IO-Link Port 2 - Output data word 15 (INT bit10)
           TBEN_L4_8IOL:O.Data[33].11   // IO-Link Port 2 - Output data word 15 (INT bit11)
           TBEN_L4_8IOL:O.Data[33].12   // IO-Link Port 2 - Output data word 15 (INT bit12)
           TBEN_L4_8IOL:O.Data[33].13   // IO-Link Port 2 - Output data word 15 (INT bit13)
           TBEN_L4_8IOL:O.Data[33].14   // IO-Link Port 2 - Output data word 15 (INT bit14)
           TBEN_L4_8IOL:O.Data[33].15   // IO-Link Port 2 - Output data word 15 (INT bit15)
           TBEN_L4_8IOL:O.Data[33].2   // IO-Link Port 2 - Output data word 15 (INT bit2)
           TBEN_L4_8IOL:O.Data[33].3   // IO-Link Port 2 - Output data word 15 (INT bit3)
           TBEN_L4_8IOL:O.Data[33].4   // IO-Link Port 2 - Output data word 15 (INT bit4)
           TBEN_L4_8IOL:O.Data[33].5   // IO-Link Port 2 - Output data word 15 (INT bit5)
           TBEN_L4_8IOL:O.Data[33].6   // IO-Link Port 2 - Output data word 15 (INT bit6)
           TBEN_L4_8IOL:O.Data[33].7   // IO-Link Port 2 - Output data word 15 (INT bit7)
           TBEN_L4_8IOL:O.Data[33].8   // IO-Link Port 2 - Output data word 15 (INT bit8)
           TBEN_L4_8IOL:O.Data[33].9   // IO-Link Port 2 - Output data word 15 (INT bit9)
           TBEN_L4_8IOL:O.Data[34]   // IO-Link Port 3 - Output data word 0
           TBEN_L4_8IOL:O.Data[34].0   // IO-Link Port 3 - Output data word 0 (INT bit0)
           TBEN_L4_8IOL:O.Data[34].1   // IO-Link Port 3 - Output data word 0 (INT bit1)
           TBEN_L4_8IOL:O.Data[34].10   // IO-Link Port 3 - Output data word 0 (INT bit10)
           TBEN_L4_8IOL:O.Data[34].11   // IO-Link Port 3 - Output data word 0 (INT bit11)
           TBEN_L4_8IOL:O.Data[34].12   // IO-Link Port 3 - Output data word 0 (INT bit12)
           TBEN_L4_8IOL:O.Data[34].13   // IO-Link Port 3 - Output data word 0 (INT bit13)
           TBEN_L4_8IOL:O.Data[34].14   // IO-Link Port 3 - Output data word 0 (INT bit14)
           TBEN_L4_8IOL:O.Data[34].15   // IO-Link Port 3 - Output data word 0 (INT bit15)
           TBEN_L4_8IOL:O.Data[34].2   // IO-Link Port 3 - Output data word 0 (INT bit2)
           TBEN_L4_8IOL:O.Data[34].3   // IO-Link Port 3 - Output data word 0 (INT bit3)
           TBEN_L4_8IOL:O.Data[34].4   // IO-Link Port 3 - Output data word 0 (INT bit4)
           TBEN_L4_8IOL:O.Data[34].5   // IO-Link Port 3 - Output data word 0 (INT bit5)
           TBEN_L4_8IOL:O.Data[34].6   // IO-Link Port 3 - Output data word 0 (INT bit6)
           TBEN_L4_8IOL:O.Data[34].7   // IO-Link Port 3 - Output data word 0 (INT bit7)
           TBEN_L4_8IOL:O.Data[34].8   // IO-Link Port 3 - Output data word 0 (INT bit8)
           TBEN_L4_8IOL:O.Data[34].9   // IO-Link Port 3 - Output data word 0 (INT bit9)
           TBEN_L4_8IOL:O.Data[35]   // IO-Link Port 3 - Output data word 1
           TBEN_L4_8IOL:O.Data[35].0   // IO-Link Port 3 - Output data word 1 (INT bit0)
           TBEN_L4_8IOL:O.Data[35].1   // IO-Link Port 3 - Output data word 1 (INT bit1)
           TBEN_L4_8IOL:O.Data[35].10   // IO-Link Port 3 - Output data word 1 (INT bit10)
           TBEN_L4_8IOL:O.Data[35].11   // IO-Link Port 3 - Output data word 1 (INT bit11)
           TBEN_L4_8IOL:O.Data[35].12   // IO-Link Port 3 - Output data word 1 (INT bit12)
           TBEN_L4_8IOL:O.Data[35].13   // IO-Link Port 3 - Output data word 1 (INT bit13)
           TBEN_L4_8IOL:O.Data[35].14   // IO-Link Port 3 - Output data word 1 (INT bit14)
           TBEN_L4_8IOL:O.Data[35].15   // IO-Link Port 3 - Output data word 1 (INT bit15)
           TBEN_L4_8IOL:O.Data[35].2   // IO-Link Port 3 - Output data word 1 (INT bit2)
           TBEN_L4_8IOL:O.Data[35].3   // IO-Link Port 3 - Output data word 1 (INT bit3)
           TBEN_L4_8IOL:O.Data[35].4   // IO-Link Port 3 - Output data word 1 (INT bit4)
           TBEN_L4_8IOL:O.Data[35].5   // IO-Link Port 3 - Output data word 1 (INT bit5)
           TBEN_L4_8IOL:O.Data[35].6   // IO-Link Port 3 - Output data word 1 (INT bit6)
           TBEN_L4_8IOL:O.Data[35].7   // IO-Link Port 3 - Output data word 1 (INT bit7)
           TBEN_L4_8IOL:O.Data[35].8   // IO-Link Port 3 - Output data word 1 (INT bit8)
           TBEN_L4_8IOL:O.Data[35].9   // IO-Link Port 3 - Output data word 1 (INT bit9)
           TBEN_L4_8IOL:O.Data[36]   // IO-Link Port 3 - Output data word 2
           TBEN_L4_8IOL:O.Data[36].0   // IO-Link Port 3 - Output data word 2 (INT bit0)
           TBEN_L4_8IOL:O.Data[36].1   // IO-Link Port 3 - Output data word 2 (INT bit1)
           TBEN_L4_8IOL:O.Data[36].10   // IO-Link Port 3 - Output data word 2 (INT bit10)
           TBEN_L4_8IOL:O.Data[36].11   // IO-Link Port 3 - Output data word 2 (INT bit11)
           TBEN_L4_8IOL:O.Data[36].12   // IO-Link Port 3 - Output data word 2 (INT bit12)
           TBEN_L4_8IOL:O.Data[36].13   // IO-Link Port 3 - Output data word 2 (INT bit13)
           TBEN_L4_8IOL:O.Data[36].14   // IO-Link Port 3 - Output data word 2 (INT bit14)
           TBEN_L4_8IOL:O.Data[36].15   // IO-Link Port 3 - Output data word 2 (INT bit15)
           TBEN_L4_8IOL:O.Data[36].2   // IO-Link Port 3 - Output data word 2 (INT bit2)
           TBEN_L4_8IOL:O.Data[36].3   // IO-Link Port 3 - Output data word 2 (INT bit3)
           TBEN_L4_8IOL:O.Data[36].4   // IO-Link Port 3 - Output data word 2 (INT bit4)
           TBEN_L4_8IOL:O.Data[36].5   // IO-Link Port 3 - Output data word 2 (INT bit5)
           TBEN_L4_8IOL:O.Data[36].6   // IO-Link Port 3 - Output data word 2 (INT bit6)
           TBEN_L4_8IOL:O.Data[36].7   // IO-Link Port 3 - Output data word 2 (INT bit7)
           TBEN_L4_8IOL:O.Data[36].8   // IO-Link Port 3 - Output data word 2 (INT bit8)
           TBEN_L4_8IOL:O.Data[36].9   // IO-Link Port 3 - Output data word 2 (INT bit9)
           TBEN_L4_8IOL:O.Data[37]   // IO-Link Port 3 - Output data word 3
           TBEN_L4_8IOL:O.Data[37].0   // IO-Link Port 3 - Output data word 3 (INT bit0)
           TBEN_L4_8IOL:O.Data[37].1   // IO-Link Port 3 - Output data word 3 (INT bit1)
           TBEN_L4_8IOL:O.Data[37].10   // IO-Link Port 3 - Output data word 3 (INT bit10)
           TBEN_L4_8IOL:O.Data[37].11   // IO-Link Port 3 - Output data word 3 (INT bit11)
           TBEN_L4_8IOL:O.Data[37].12   // IO-Link Port 3 - Output data word 3 (INT bit12)
           TBEN_L4_8IOL:O.Data[37].13   // IO-Link Port 3 - Output data word 3 (INT bit13)
           TBEN_L4_8IOL:O.Data[37].14   // IO-Link Port 3 - Output data word 3 (INT bit14)
           TBEN_L4_8IOL:O.Data[37].15   // IO-Link Port 3 - Output data word 3 (INT bit15)
           TBEN_L4_8IOL:O.Data[37].2   // IO-Link Port 3 - Output data word 3 (INT bit2)
           TBEN_L4_8IOL:O.Data[37].3   // IO-Link Port 3 - Output data word 3 (INT bit3)
           TBEN_L4_8IOL:O.Data[37].4   // IO-Link Port 3 - Output data word 3 (INT bit4)
           TBEN_L4_8IOL:O.Data[37].5   // IO-Link Port 3 - Output data word 3 (INT bit5)
           TBEN_L4_8IOL:O.Data[37].6   // IO-Link Port 3 - Output data word 3 (INT bit6)
           TBEN_L4_8IOL:O.Data[37].7   // IO-Link Port 3 - Output data word 3 (INT bit7)
           TBEN_L4_8IOL:O.Data[37].8   // IO-Link Port 3 - Output data word 3 (INT bit8)
           TBEN_L4_8IOL:O.Data[37].9   // IO-Link Port 3 - Output data word 3 (INT bit9)
           TBEN_L4_8IOL:O.Data[38]   // IO-Link Port 3 - Output data word 4
           TBEN_L4_8IOL:O.Data[38].0   // IO-Link Port 3 - Output data word 4 (INT bit0)
           TBEN_L4_8IOL:O.Data[38].1   // IO-Link Port 3 - Output data word 4 (INT bit1)
           TBEN_L4_8IOL:O.Data[38].10   // IO-Link Port 3 - Output data word 4 (INT bit10)
           TBEN_L4_8IOL:O.Data[38].11   // IO-Link Port 3 - Output data word 4 (INT bit11)
           TBEN_L4_8IOL:O.Data[38].12   // IO-Link Port 3 - Output data word 4 (INT bit12)
           TBEN_L4_8IOL:O.Data[38].13   // IO-Link Port 3 - Output data word 4 (INT bit13)
           TBEN_L4_8IOL:O.Data[38].14   // IO-Link Port 3 - Output data word 4 (INT bit14)
           TBEN_L4_8IOL:O.Data[38].15   // IO-Link Port 3 - Output data word 4 (INT bit15)
           TBEN_L4_8IOL:O.Data[38].2   // IO-Link Port 3 - Output data word 4 (INT bit2)
           TBEN_L4_8IOL:O.Data[38].3   // IO-Link Port 3 - Output data word 4 (INT bit3)
           TBEN_L4_8IOL:O.Data[38].4   // IO-Link Port 3 - Output data word 4 (INT bit4)
           TBEN_L4_8IOL:O.Data[38].5   // IO-Link Port 3 - Output data word 4 (INT bit5)
           TBEN_L4_8IOL:O.Data[38].6   // IO-Link Port 3 - Output data word 4 (INT bit6)
           TBEN_L4_8IOL:O.Data[38].7   // IO-Link Port 3 - Output data word 4 (INT bit7)
           TBEN_L4_8IOL:O.Data[38].8   // IO-Link Port 3 - Output data word 4 (INT bit8)
           TBEN_L4_8IOL:O.Data[38].9   // IO-Link Port 3 - Output data word 4 (INT bit9)
           TBEN_L4_8IOL:O.Data[39]   // IO-Link Port 3 - Output data word 5
           TBEN_L4_8IOL:O.Data[39].0   // IO-Link Port 3 - Output data word 5 (INT bit0)
           TBEN_L4_8IOL:O.Data[39].1   // IO-Link Port 3 - Output data word 5 (INT bit1)
           TBEN_L4_8IOL:O.Data[39].10   // IO-Link Port 3 - Output data word 5 (INT bit10)
           TBEN_L4_8IOL:O.Data[39].11   // IO-Link Port 3 - Output data word 5 (INT bit11)
           TBEN_L4_8IOL:O.Data[39].12   // IO-Link Port 3 - Output data word 5 (INT bit12)
           TBEN_L4_8IOL:O.Data[39].13   // IO-Link Port 3 - Output data word 5 (INT bit13)
           TBEN_L4_8IOL:O.Data[39].14   // IO-Link Port 3 - Output data word 5 (INT bit14)
           TBEN_L4_8IOL:O.Data[39].15   // IO-Link Port 3 - Output data word 5 (INT bit15)
           TBEN_L4_8IOL:O.Data[39].2   // IO-Link Port 3 - Output data word 5 (INT bit2)
           TBEN_L4_8IOL:O.Data[39].3   // IO-Link Port 3 - Output data word 5 (INT bit3)
           TBEN_L4_8IOL:O.Data[39].4   // IO-Link Port 3 - Output data word 5 (INT bit4)
           TBEN_L4_8IOL:O.Data[39].5   // IO-Link Port 3 - Output data word 5 (INT bit5)
           TBEN_L4_8IOL:O.Data[39].6   // IO-Link Port 3 - Output data word 5 (INT bit6)
           TBEN_L4_8IOL:O.Data[39].7   // IO-Link Port 3 - Output data word 5 (INT bit7)
           TBEN_L4_8IOL:O.Data[39].8   // IO-Link Port 3 - Output data word 5 (INT bit8)
           TBEN_L4_8IOL:O.Data[39].9   // IO-Link Port 3 - Output data word 5 (INT bit9)
           TBEN_L4_8IOL:O.Data[3]   // IO-Link Port 1 - Output data word 1
           TBEN_L4_8IOL:O.Data[3].0   // IO-Link Port 1 - Output data word 1 (INT bit0)
           TBEN_L4_8IOL:O.Data[3].1   // IO-Link Port 1 - Output data word 1 (INT bit1)
           TBEN_L4_8IOL:O.Data[3].10   // IO-Link Port 1 - Output data word 1 (INT bit10)
           TBEN_L4_8IOL:O.Data[3].11   // IO-Link Port 1 - Output data word 1 (INT bit11)
           TBEN_L4_8IOL:O.Data[3].12   // IO-Link Port 1 - Output data word 1 (INT bit12)
           TBEN_L4_8IOL:O.Data[3].13   // IO-Link Port 1 - Output data word 1 (INT bit13)
           TBEN_L4_8IOL:O.Data[3].14   // IO-Link Port 1 - Output data word 1 (INT bit14)
           TBEN_L4_8IOL:O.Data[3].15   // IO-Link Port 1 - Output data word 1 (INT bit15)
           TBEN_L4_8IOL:O.Data[3].2   // IO-Link Port 1 - Output data word 1 (INT bit2)
           TBEN_L4_8IOL:O.Data[3].3   // IO-Link Port 1 - Output data word 1 (INT bit3)
           TBEN_L4_8IOL:O.Data[3].4   // IO-Link Port 1 - Output data word 1 (INT bit4)
           TBEN_L4_8IOL:O.Data[3].5   // IO-Link Port 1 - Output data word 1 (INT bit5)
           TBEN_L4_8IOL:O.Data[3].6   // IO-Link Port 1 - Output data word 1 (INT bit6)
           TBEN_L4_8IOL:O.Data[3].7   // IO-Link Port 1 - Output data word 1 (INT bit7)
           TBEN_L4_8IOL:O.Data[3].8   // IO-Link Port 1 - Output data word 1 (INT bit8)
           TBEN_L4_8IOL:O.Data[3].9   // IO-Link Port 1 - Output data word 1 (INT bit9)
           TBEN_L4_8IOL:O.Data[40]   // IO-Link Port 3 - Output data word 6
           TBEN_L4_8IOL:O.Data[40].0   // IO-Link Port 3 - Output data word 6 (INT bit0)
           TBEN_L4_8IOL:O.Data[40].1   // IO-Link Port 3 - Output data word 6 (INT bit1)
           TBEN_L4_8IOL:O.Data[40].10   // IO-Link Port 3 - Output data word 6 (INT bit10)
           TBEN_L4_8IOL:O.Data[40].11   // IO-Link Port 3 - Output data word 6 (INT bit11)
           TBEN_L4_8IOL:O.Data[40].12   // IO-Link Port 3 - Output data word 6 (INT bit12)
           TBEN_L4_8IOL:O.Data[40].13   // IO-Link Port 3 - Output data word 6 (INT bit13)
           TBEN_L4_8IOL:O.Data[40].14   // IO-Link Port 3 - Output data word 6 (INT bit14)
           TBEN_L4_8IOL:O.Data[40].15   // IO-Link Port 3 - Output data word 6 (INT bit15)
           TBEN_L4_8IOL:O.Data[40].2   // IO-Link Port 3 - Output data word 6 (INT bit2)
           TBEN_L4_8IOL:O.Data[40].3   // IO-Link Port 3 - Output data word 6 (INT bit3)
           TBEN_L4_8IOL:O.Data[40].4   // IO-Link Port 3 - Output data word 6 (INT bit4)
           TBEN_L4_8IOL:O.Data[40].5   // IO-Link Port 3 - Output data word 6 (INT bit5)
           TBEN_L4_8IOL:O.Data[40].6   // IO-Link Port 3 - Output data word 6 (INT bit6)
           TBEN_L4_8IOL:O.Data[40].7   // IO-Link Port 3 - Output data word 6 (INT bit7)
           TBEN_L4_8IOL:O.Data[40].8   // IO-Link Port 3 - Output data word 6 (INT bit8)
           TBEN_L4_8IOL:O.Data[40].9   // IO-Link Port 3 - Output data word 6 (INT bit9)
           TBEN_L4_8IOL:O.Data[41]   // IO-Link Port 3 - Output data word 7
           TBEN_L4_8IOL:O.Data[41].0   // IO-Link Port 3 - Output data word 7 (INT bit0)
           TBEN_L4_8IOL:O.Data[41].1   // IO-Link Port 3 - Output data word 7 (INT bit1)
           TBEN_L4_8IOL:O.Data[41].10   // IO-Link Port 3 - Output data word 7 (INT bit10)
           TBEN_L4_8IOL:O.Data[41].11   // IO-Link Port 3 - Output data word 7 (INT bit11)
           TBEN_L4_8IOL:O.Data[41].12   // IO-Link Port 3 - Output data word 7 (INT bit12)
           TBEN_L4_8IOL:O.Data[41].13   // IO-Link Port 3 - Output data word 7 (INT bit13)
           TBEN_L4_8IOL:O.Data[41].14   // IO-Link Port 3 - Output data word 7 (INT bit14)
           TBEN_L4_8IOL:O.Data[41].15   // IO-Link Port 3 - Output data word 7 (INT bit15)
           TBEN_L4_8IOL:O.Data[41].2   // IO-Link Port 3 - Output data word 7 (INT bit2)
           TBEN_L4_8IOL:O.Data[41].3   // IO-Link Port 3 - Output data word 7 (INT bit3)
           TBEN_L4_8IOL:O.Data[41].4   // IO-Link Port 3 - Output data word 7 (INT bit4)
           TBEN_L4_8IOL:O.Data[41].5   // IO-Link Port 3 - Output data word 7 (INT bit5)
           TBEN_L4_8IOL:O.Data[41].6   // IO-Link Port 3 - Output data word 7 (INT bit6)
           TBEN_L4_8IOL:O.Data[41].7   // IO-Link Port 3 - Output data word 7 (INT bit7)
           TBEN_L4_8IOL:O.Data[41].8   // IO-Link Port 3 - Output data word 7 (INT bit8)
           TBEN_L4_8IOL:O.Data[41].9   // IO-Link Port 3 - Output data word 7 (INT bit9)
           TBEN_L4_8IOL:O.Data[42]   // IO-Link Port 3 - Output data word 8
           TBEN_L4_8IOL:O.Data[42].0   // IO-Link Port 3 - Output data word 8 (INT bit0)
           TBEN_L4_8IOL:O.Data[42].1   // IO-Link Port 3 - Output data word 8 (INT bit1)
           TBEN_L4_8IOL:O.Data[42].10   // IO-Link Port 3 - Output data word 8 (INT bit10)
           TBEN_L4_8IOL:O.Data[42].11   // IO-Link Port 3 - Output data word 8 (INT bit11)
           TBEN_L4_8IOL:O.Data[42].12   // IO-Link Port 3 - Output data word 8 (INT bit12)
           TBEN_L4_8IOL:O.Data[42].13   // IO-Link Port 3 - Output data word 8 (INT bit13)
           TBEN_L4_8IOL:O.Data[42].14   // IO-Link Port 3 - Output data word 8 (INT bit14)
           TBEN_L4_8IOL:O.Data[42].15   // IO-Link Port 3 - Output data word 8 (INT bit15)
           TBEN_L4_8IOL:O.Data[42].2   // IO-Link Port 3 - Output data word 8 (INT bit2)
           TBEN_L4_8IOL:O.Data[42].3   // IO-Link Port 3 - Output data word 8 (INT bit3)
           TBEN_L4_8IOL:O.Data[42].4   // IO-Link Port 3 - Output data word 8 (INT bit4)
           TBEN_L4_8IOL:O.Data[42].5   // IO-Link Port 3 - Output data word 8 (INT bit5)
           TBEN_L4_8IOL:O.Data[42].6   // IO-Link Port 3 - Output data word 8 (INT bit6)
           TBEN_L4_8IOL:O.Data[42].7   // IO-Link Port 3 - Output data word 8 (INT bit7)
           TBEN_L4_8IOL:O.Data[42].8   // IO-Link Port 3 - Output data word 8 (INT bit8)
           TBEN_L4_8IOL:O.Data[42].9   // IO-Link Port 3 - Output data word 8 (INT bit9)
           TBEN_L4_8IOL:O.Data[43]   // IO-Link Port 3 - Output data word 9
           TBEN_L4_8IOL:O.Data[43].0   // IO-Link Port 3 - Output data word 9 (INT bit0)
           TBEN_L4_8IOL:O.Data[43].1   // IO-Link Port 3 - Output data word 9 (INT bit1)
           TBEN_L4_8IOL:O.Data[43].10   // IO-Link Port 3 - Output data word 9 (INT bit10)
           TBEN_L4_8IOL:O.Data[43].11   // IO-Link Port 3 - Output data word 9 (INT bit11)
           TBEN_L4_8IOL:O.Data[43].12   // IO-Link Port 3 - Output data word 9 (INT bit12)
           TBEN_L4_8IOL:O.Data[43].13   // IO-Link Port 3 - Output data word 9 (INT bit13)
           TBEN_L4_8IOL:O.Data[43].14   // IO-Link Port 3 - Output data word 9 (INT bit14)
           TBEN_L4_8IOL:O.Data[43].15   // IO-Link Port 3 - Output data word 9 (INT bit15)
           TBEN_L4_8IOL:O.Data[43].2   // IO-Link Port 3 - Output data word 9 (INT bit2)
           TBEN_L4_8IOL:O.Data[43].3   // IO-Link Port 3 - Output data word 9 (INT bit3)
           TBEN_L4_8IOL:O.Data[43].4   // IO-Link Port 3 - Output data word 9 (INT bit4)
           TBEN_L4_8IOL:O.Data[43].5   // IO-Link Port 3 - Output data word 9 (INT bit5)
           TBEN_L4_8IOL:O.Data[43].6   // IO-Link Port 3 - Output data word 9 (INT bit6)
           TBEN_L4_8IOL:O.Data[43].7   // IO-Link Port 3 - Output data word 9 (INT bit7)
           TBEN_L4_8IOL:O.Data[43].8   // IO-Link Port 3 - Output data word 9 (INT bit8)
           TBEN_L4_8IOL:O.Data[43].9   // IO-Link Port 3 - Output data word 9 (INT bit9)
           TBEN_L4_8IOL:O.Data[44]   // IO-Link Port 3 - Output data word 10
           TBEN_L4_8IOL:O.Data[44].0   // IO-Link Port 3 - Output data word 10 (INT bit0)
           TBEN_L4_8IOL:O.Data[44].1   // IO-Link Port 3 - Output data word 10 (INT bit1)
           TBEN_L4_8IOL:O.Data[44].10   // IO-Link Port 3 - Output data word 10 (INT bit10)
           TBEN_L4_8IOL:O.Data[44].11   // IO-Link Port 3 - Output data word 10 (INT bit11)
           TBEN_L4_8IOL:O.Data[44].12   // IO-Link Port 3 - Output data word 10 (INT bit12)
           TBEN_L4_8IOL:O.Data[44].13   // IO-Link Port 3 - Output data word 10 (INT bit13)
           TBEN_L4_8IOL:O.Data[44].14   // IO-Link Port 3 - Output data word 10 (INT bit14)
           TBEN_L4_8IOL:O.Data[44].15   // IO-Link Port 3 - Output data word 10 (INT bit15)
           TBEN_L4_8IOL:O.Data[44].2   // IO-Link Port 3 - Output data word 10 (INT bit2)
           TBEN_L4_8IOL:O.Data[44].3   // IO-Link Port 3 - Output data word 10 (INT bit3)
           TBEN_L4_8IOL:O.Data[44].4   // IO-Link Port 3 - Output data word 10 (INT bit4)
           TBEN_L4_8IOL:O.Data[44].5   // IO-Link Port 3 - Output data word 10 (INT bit5)
           TBEN_L4_8IOL:O.Data[44].6   // IO-Link Port 3 - Output data word 10 (INT bit6)
           TBEN_L4_8IOL:O.Data[44].7   // IO-Link Port 3 - Output data word 10 (INT bit7)
           TBEN_L4_8IOL:O.Data[44].8   // IO-Link Port 3 - Output data word 10 (INT bit8)
           TBEN_L4_8IOL:O.Data[44].9   // IO-Link Port 3 - Output data word 10 (INT bit9)
           TBEN_L4_8IOL:O.Data[45]   // IO-Link Port 3 - Output data word 11
           TBEN_L4_8IOL:O.Data[45].0   // IO-Link Port 3 - Output data word 11 (INT bit0)
           TBEN_L4_8IOL:O.Data[45].1   // IO-Link Port 3 - Output data word 11 (INT bit1)
           TBEN_L4_8IOL:O.Data[45].10   // IO-Link Port 3 - Output data word 11 (INT bit10)
           TBEN_L4_8IOL:O.Data[45].11   // IO-Link Port 3 - Output data word 11 (INT bit11)
           TBEN_L4_8IOL:O.Data[45].12   // IO-Link Port 3 - Output data word 11 (INT bit12)
           TBEN_L4_8IOL:O.Data[45].13   // IO-Link Port 3 - Output data word 11 (INT bit13)
           TBEN_L4_8IOL:O.Data[45].14   // IO-Link Port 3 - Output data word 11 (INT bit14)
           TBEN_L4_8IOL:O.Data[45].15   // IO-Link Port 3 - Output data word 11 (INT bit15)
           TBEN_L4_8IOL:O.Data[45].2   // IO-Link Port 3 - Output data word 11 (INT bit2)
           TBEN_L4_8IOL:O.Data[45].3   // IO-Link Port 3 - Output data word 11 (INT bit3)
           TBEN_L4_8IOL:O.Data[45].4   // IO-Link Port 3 - Output data word 11 (INT bit4)
           TBEN_L4_8IOL:O.Data[45].5   // IO-Link Port 3 - Output data word 11 (INT bit5)
           TBEN_L4_8IOL:O.Data[45].6   // IO-Link Port 3 - Output data word 11 (INT bit6)
           TBEN_L4_8IOL:O.Data[45].7   // IO-Link Port 3 - Output data word 11 (INT bit7)
           TBEN_L4_8IOL:O.Data[45].8   // IO-Link Port 3 - Output data word 11 (INT bit8)
           TBEN_L4_8IOL:O.Data[45].9   // IO-Link Port 3 - Output data word 11 (INT bit9)
           TBEN_L4_8IOL:O.Data[46]   // IO-Link Port 3 - Output data word 12
           TBEN_L4_8IOL:O.Data[46].0   // IO-Link Port 3 - Output data word 12 (INT bit0)
           TBEN_L4_8IOL:O.Data[46].1   // IO-Link Port 3 - Output data word 12 (INT bit1)
           TBEN_L4_8IOL:O.Data[46].10   // IO-Link Port 3 - Output data word 12 (INT bit10)
           TBEN_L4_8IOL:O.Data[46].11   // IO-Link Port 3 - Output data word 12 (INT bit11)
           TBEN_L4_8IOL:O.Data[46].12   // IO-Link Port 3 - Output data word 12 (INT bit12)
           TBEN_L4_8IOL:O.Data[46].13   // IO-Link Port 3 - Output data word 12 (INT bit13)
           TBEN_L4_8IOL:O.Data[46].14   // IO-Link Port 3 - Output data word 12 (INT bit14)
           TBEN_L4_8IOL:O.Data[46].15   // IO-Link Port 3 - Output data word 12 (INT bit15)
           TBEN_L4_8IOL:O.Data[46].2   // IO-Link Port 3 - Output data word 12 (INT bit2)
           TBEN_L4_8IOL:O.Data[46].3   // IO-Link Port 3 - Output data word 12 (INT bit3)
           TBEN_L4_8IOL:O.Data[46].4   // IO-Link Port 3 - Output data word 12 (INT bit4)
           TBEN_L4_8IOL:O.Data[46].5   // IO-Link Port 3 - Output data word 12 (INT bit5)
           TBEN_L4_8IOL:O.Data[46].6   // IO-Link Port 3 - Output data word 12 (INT bit6)
           TBEN_L4_8IOL:O.Data[46].7   // IO-Link Port 3 - Output data word 12 (INT bit7)
           TBEN_L4_8IOL:O.Data[46].8   // IO-Link Port 3 - Output data word 12 (INT bit8)
           TBEN_L4_8IOL:O.Data[46].9   // IO-Link Port 3 - Output data word 12 (INT bit9)
           TBEN_L4_8IOL:O.Data[47]   // IO-Link Port 3 - Output data word 13
           TBEN_L4_8IOL:O.Data[47].0   // IO-Link Port 3 - Output data word 13 (INT bit0)
           TBEN_L4_8IOL:O.Data[47].1   // IO-Link Port 3 - Output data word 13 (INT bit1)
           TBEN_L4_8IOL:O.Data[47].10   // IO-Link Port 3 - Output data word 13 (INT bit10)
           TBEN_L4_8IOL:O.Data[47].11   // IO-Link Port 3 - Output data word 13 (INT bit11)
           TBEN_L4_8IOL:O.Data[47].12   // IO-Link Port 3 - Output data word 13 (INT bit12)
           TBEN_L4_8IOL:O.Data[47].13   // IO-Link Port 3 - Output data word 13 (INT bit13)
           TBEN_L4_8IOL:O.Data[47].14   // IO-Link Port 3 - Output data word 13 (INT bit14)
           TBEN_L4_8IOL:O.Data[47].15   // IO-Link Port 3 - Output data word 13 (INT bit15)
           TBEN_L4_8IOL:O.Data[47].2   // IO-Link Port 3 - Output data word 13 (INT bit2)
           TBEN_L4_8IOL:O.Data[47].3   // IO-Link Port 3 - Output data word 13 (INT bit3)
           TBEN_L4_8IOL:O.Data[47].4   // IO-Link Port 3 - Output data word 13 (INT bit4)
           TBEN_L4_8IOL:O.Data[47].5   // IO-Link Port 3 - Output data word 13 (INT bit5)
           TBEN_L4_8IOL:O.Data[47].6   // IO-Link Port 3 - Output data word 13 (INT bit6)
           TBEN_L4_8IOL:O.Data[47].7   // IO-Link Port 3 - Output data word 13 (INT bit7)
           TBEN_L4_8IOL:O.Data[47].8   // IO-Link Port 3 - Output data word 13 (INT bit8)
           TBEN_L4_8IOL:O.Data[47].9   // IO-Link Port 3 - Output data word 13 (INT bit9)
           TBEN_L4_8IOL:O.Data[48]   // IO-Link Port 3 - Output data word 14
           TBEN_L4_8IOL:O.Data[48].0   // IO-Link Port 3 - Output data word 14 (INT bit0)
           TBEN_L4_8IOL:O.Data[48].1   // IO-Link Port 3 - Output data word 14 (INT bit1)
           TBEN_L4_8IOL:O.Data[48].10   // IO-Link Port 3 - Output data word 14 (INT bit10)
           TBEN_L4_8IOL:O.Data[48].11   // IO-Link Port 3 - Output data word 14 (INT bit11)
           TBEN_L4_8IOL:O.Data[48].12   // IO-Link Port 3 - Output data word 14 (INT bit12)
           TBEN_L4_8IOL:O.Data[48].13   // IO-Link Port 3 - Output data word 14 (INT bit13)
           TBEN_L4_8IOL:O.Data[48].14   // IO-Link Port 3 - Output data word 14 (INT bit14)
           TBEN_L4_8IOL:O.Data[48].15   // IO-Link Port 3 - Output data word 14 (INT bit15)
           TBEN_L4_8IOL:O.Data[48].2   // IO-Link Port 3 - Output data word 14 (INT bit2)
           TBEN_L4_8IOL:O.Data[48].3   // IO-Link Port 3 - Output data word 14 (INT bit3)
           TBEN_L4_8IOL:O.Data[48].4   // IO-Link Port 3 - Output data word 14 (INT bit4)
           TBEN_L4_8IOL:O.Data[48].5   // IO-Link Port 3 - Output data word 14 (INT bit5)
           TBEN_L4_8IOL:O.Data[48].6   // IO-Link Port 3 - Output data word 14 (INT bit6)
           TBEN_L4_8IOL:O.Data[48].7   // IO-Link Port 3 - Output data word 14 (INT bit7)
           TBEN_L4_8IOL:O.Data[48].8   // IO-Link Port 3 - Output data word 14 (INT bit8)
           TBEN_L4_8IOL:O.Data[48].9   // IO-Link Port 3 - Output data word 14 (INT bit9)
           TBEN_L4_8IOL:O.Data[49]   // IO-Link Port 3 - Output data word 15
           TBEN_L4_8IOL:O.Data[49].0   // IO-Link Port 3 - Output data word 15 (INT bit0)
           TBEN_L4_8IOL:O.Data[49].1   // IO-Link Port 3 - Output data word 15 (INT bit1)
           TBEN_L4_8IOL:O.Data[49].10   // IO-Link Port 3 - Output data word 15 (INT bit10)
           TBEN_L4_8IOL:O.Data[49].11   // IO-Link Port 3 - Output data word 15 (INT bit11)
           TBEN_L4_8IOL:O.Data[49].12   // IO-Link Port 3 - Output data word 15 (INT bit12)
           TBEN_L4_8IOL:O.Data[49].13   // IO-Link Port 3 - Output data word 15 (INT bit13)
           TBEN_L4_8IOL:O.Data[49].14   // IO-Link Port 3 - Output data word 15 (INT bit14)
           TBEN_L4_8IOL:O.Data[49].15   // IO-Link Port 3 - Output data word 15 (INT bit15)
           TBEN_L4_8IOL:O.Data[49].2   // IO-Link Port 3 - Output data word 15 (INT bit2)
           TBEN_L4_8IOL:O.Data[49].3   // IO-Link Port 3 - Output data word 15 (INT bit3)
           TBEN_L4_8IOL:O.Data[49].4   // IO-Link Port 3 - Output data word 15 (INT bit4)
           TBEN_L4_8IOL:O.Data[49].5   // IO-Link Port 3 - Output data word 15 (INT bit5)
           TBEN_L4_8IOL:O.Data[49].6   // IO-Link Port 3 - Output data word 15 (INT bit6)
           TBEN_L4_8IOL:O.Data[49].7   // IO-Link Port 3 - Output data word 15 (INT bit7)
           TBEN_L4_8IOL:O.Data[49].8   // IO-Link Port 3 - Output data word 15 (INT bit8)
           TBEN_L4_8IOL:O.Data[49].9   // IO-Link Port 3 - Output data word 15 (INT bit9)
           TBEN_L4_8IOL:O.Data[4]   // IO-Link Port 1 - Output data word 2
           TBEN_L4_8IOL:O.Data[4].0   // IO-Link Port 1 - Output data word 2 (INT bit0)
           TBEN_L4_8IOL:O.Data[4].1   // IO-Link Port 1 - Output data word 2 (INT bit1)
           TBEN_L4_8IOL:O.Data[4].10   // IO-Link Port 1 - Output data word 2 (INT bit10)
           TBEN_L4_8IOL:O.Data[4].11   // IO-Link Port 1 - Output data word 2 (INT bit11)
           TBEN_L4_8IOL:O.Data[4].12   // IO-Link Port 1 - Output data word 2 (INT bit12)
           TBEN_L4_8IOL:O.Data[4].13   // IO-Link Port 1 - Output data word 2 (INT bit13)
           TBEN_L4_8IOL:O.Data[4].14   // IO-Link Port 1 - Output data word 2 (INT bit14)
           TBEN_L4_8IOL:O.Data[4].15   // IO-Link Port 1 - Output data word 2 (INT bit15)
           TBEN_L4_8IOL:O.Data[4].2   // IO-Link Port 1 - Output data word 2 (INT bit2)
           TBEN_L4_8IOL:O.Data[4].3   // IO-Link Port 1 - Output data word 2 (INT bit3)
           TBEN_L4_8IOL:O.Data[4].4   // IO-Link Port 1 - Output data word 2 (INT bit4)
           TBEN_L4_8IOL:O.Data[4].5   // IO-Link Port 1 - Output data word 2 (INT bit5)
           TBEN_L4_8IOL:O.Data[4].6   // IO-Link Port 1 - Output data word 2 (INT bit6)
           TBEN_L4_8IOL:O.Data[4].7   // IO-Link Port 1 - Output data word 2 (INT bit7)
           TBEN_L4_8IOL:O.Data[4].8   // IO-Link Port 1 - Output data word 2 (INT bit8)
           TBEN_L4_8IOL:O.Data[4].9   // IO-Link Port 1 - Output data word 2 (INT bit9)
           TBEN_L4_8IOL:O.Data[50]   // IO-Link Port 4 - Output data word 0
           TBEN_L4_8IOL:O.Data[50].0   // IO-Link Port 4 - Output data word 0 (INT bit0)
           TBEN_L4_8IOL:O.Data[50].1   // IO-Link Port 4 - Output data word 0 (INT bit1)
           TBEN_L4_8IOL:O.Data[50].10   // IO-Link Port 4 - Output data word 0 (INT bit10)
           TBEN_L4_8IOL:O.Data[50].11   // IO-Link Port 4 - Output data word 0 (INT bit11)
           TBEN_L4_8IOL:O.Data[50].12   // IO-Link Port 4 - Output data word 0 (INT bit12)
           TBEN_L4_8IOL:O.Data[50].13   // IO-Link Port 4 - Output data word 0 (INT bit13)
           TBEN_L4_8IOL:O.Data[50].14   // IO-Link Port 4 - Output data word 0 (INT bit14)
           TBEN_L4_8IOL:O.Data[50].15   // IO-Link Port 4 - Output data word 0 (INT bit15)
           TBEN_L4_8IOL:O.Data[50].2   // IO-Link Port 4 - Output data word 0 (INT bit2)
           TBEN_L4_8IOL:O.Data[50].3   // IO-Link Port 4 - Output data word 0 (INT bit3)
           TBEN_L4_8IOL:O.Data[50].4   // IO-Link Port 4 - Output data word 0 (INT bit4)
           TBEN_L4_8IOL:O.Data[50].5   // IO-Link Port 4 - Output data word 0 (INT bit5)
           TBEN_L4_8IOL:O.Data[50].6   // IO-Link Port 4 - Output data word 0 (INT bit6)
           TBEN_L4_8IOL:O.Data[50].7   // IO-Link Port 4 - Output data word 0 (INT bit7)
           TBEN_L4_8IOL:O.Data[50].8   // IO-Link Port 4 - Output data word 0 (INT bit8)
           TBEN_L4_8IOL:O.Data[50].9   // IO-Link Port 4 - Output data word 0 (INT bit9)
           TBEN_L4_8IOL:O.Data[51]   // IO-Link Port 4 - Output data word 1
           TBEN_L4_8IOL:O.Data[51].0   // IO-Link Port 4 - Output data word 1 (INT bit0)
           TBEN_L4_8IOL:O.Data[51].1   // IO-Link Port 4 - Output data word 1 (INT bit1)
           TBEN_L4_8IOL:O.Data[51].10   // IO-Link Port 4 - Output data word 1 (INT bit10)
           TBEN_L4_8IOL:O.Data[51].11   // IO-Link Port 4 - Output data word 1 (INT bit11)
           TBEN_L4_8IOL:O.Data[51].12   // IO-Link Port 4 - Output data word 1 (INT bit12)
           TBEN_L4_8IOL:O.Data[51].13   // IO-Link Port 4 - Output data word 1 (INT bit13)
           TBEN_L4_8IOL:O.Data[51].14   // IO-Link Port 4 - Output data word 1 (INT bit14)
           TBEN_L4_8IOL:O.Data[51].15   // IO-Link Port 4 - Output data word 1 (INT bit15)
           TBEN_L4_8IOL:O.Data[51].2   // IO-Link Port 4 - Output data word 1 (INT bit2)
           TBEN_L4_8IOL:O.Data[51].3   // IO-Link Port 4 - Output data word 1 (INT bit3)
           TBEN_L4_8IOL:O.Data[51].4   // IO-Link Port 4 - Output data word 1 (INT bit4)
           TBEN_L4_8IOL:O.Data[51].5   // IO-Link Port 4 - Output data word 1 (INT bit5)
           TBEN_L4_8IOL:O.Data[51].6   // IO-Link Port 4 - Output data word 1 (INT bit6)
           TBEN_L4_8IOL:O.Data[51].7   // IO-Link Port 4 - Output data word 1 (INT bit7)
           TBEN_L4_8IOL:O.Data[51].8   // IO-Link Port 4 - Output data word 1 (INT bit8)
           TBEN_L4_8IOL:O.Data[51].9   // IO-Link Port 4 - Output data word 1 (INT bit9)
           TBEN_L4_8IOL:O.Data[52]   // IO-Link Port 4 - Output data word 2
           TBEN_L4_8IOL:O.Data[52].0   // IO-Link Port 4 - Output data word 2 (INT bit0)
           TBEN_L4_8IOL:O.Data[52].1   // IO-Link Port 4 - Output data word 2 (INT bit1)
           TBEN_L4_8IOL:O.Data[52].10   // IO-Link Port 4 - Output data word 2 (INT bit10)
           TBEN_L4_8IOL:O.Data[52].11   // IO-Link Port 4 - Output data word 2 (INT bit11)
           TBEN_L4_8IOL:O.Data[52].12   // IO-Link Port 4 - Output data word 2 (INT bit12)
           TBEN_L4_8IOL:O.Data[52].13   // IO-Link Port 4 - Output data word 2 (INT bit13)
           TBEN_L4_8IOL:O.Data[52].14   // IO-Link Port 4 - Output data word 2 (INT bit14)
           TBEN_L4_8IOL:O.Data[52].15   // IO-Link Port 4 - Output data word 2 (INT bit15)
           TBEN_L4_8IOL:O.Data[52].2   // IO-Link Port 4 - Output data word 2 (INT bit2)
           TBEN_L4_8IOL:O.Data[52].3   // IO-Link Port 4 - Output data word 2 (INT bit3)
           TBEN_L4_8IOL:O.Data[52].4   // IO-Link Port 4 - Output data word 2 (INT bit4)
           TBEN_L4_8IOL:O.Data[52].5   // IO-Link Port 4 - Output data word 2 (INT bit5)
           TBEN_L4_8IOL:O.Data[52].6   // IO-Link Port 4 - Output data word 2 (INT bit6)
           TBEN_L4_8IOL:O.Data[52].7   // IO-Link Port 4 - Output data word 2 (INT bit7)
           TBEN_L4_8IOL:O.Data[52].8   // IO-Link Port 4 - Output data word 2 (INT bit8)
           TBEN_L4_8IOL:O.Data[52].9   // IO-Link Port 4 - Output data word 2 (INT bit9)
           TBEN_L4_8IOL:O.Data[53]   // IO-Link Port 4 - Output data word 3
           TBEN_L4_8IOL:O.Data[53].0   // IO-Link Port 4 - Output data word 3 (INT bit0)
           TBEN_L4_8IOL:O.Data[53].1   // IO-Link Port 4 - Output data word 3 (INT bit1)
           TBEN_L4_8IOL:O.Data[53].10   // IO-Link Port 4 - Output data word 3 (INT bit10)
           TBEN_L4_8IOL:O.Data[53].11   // IO-Link Port 4 - Output data word 3 (INT bit11)
           TBEN_L4_8IOL:O.Data[53].12   // IO-Link Port 4 - Output data word 3 (INT bit12)
           TBEN_L4_8IOL:O.Data[53].13   // IO-Link Port 4 - Output data word 3 (INT bit13)
           TBEN_L4_8IOL:O.Data[53].14   // IO-Link Port 4 - Output data word 3 (INT bit14)
           TBEN_L4_8IOL:O.Data[53].15   // IO-Link Port 4 - Output data word 3 (INT bit15)
           TBEN_L4_8IOL:O.Data[53].2   // IO-Link Port 4 - Output data word 3 (INT bit2)
           TBEN_L4_8IOL:O.Data[53].3   // IO-Link Port 4 - Output data word 3 (INT bit3)
           TBEN_L4_8IOL:O.Data[53].4   // IO-Link Port 4 - Output data word 3 (INT bit4)
           TBEN_L4_8IOL:O.Data[53].5   // IO-Link Port 4 - Output data word 3 (INT bit5)
           TBEN_L4_8IOL:O.Data[53].6   // IO-Link Port 4 - Output data word 3 (INT bit6)
           TBEN_L4_8IOL:O.Data[53].7   // IO-Link Port 4 - Output data word 3 (INT bit7)
           TBEN_L4_8IOL:O.Data[53].8   // IO-Link Port 4 - Output data word 3 (INT bit8)
           TBEN_L4_8IOL:O.Data[53].9   // IO-Link Port 4 - Output data word 3 (INT bit9)
           TBEN_L4_8IOL:O.Data[54]   // IO-Link Port 4 - Output data word 4
           TBEN_L4_8IOL:O.Data[54].0   // IO-Link Port 4 - Output data word 4 (INT bit0)
           TBEN_L4_8IOL:O.Data[54].1   // IO-Link Port 4 - Output data word 4 (INT bit1)
           TBEN_L4_8IOL:O.Data[54].10   // IO-Link Port 4 - Output data word 4 (INT bit10)
           TBEN_L4_8IOL:O.Data[54].11   // IO-Link Port 4 - Output data word 4 (INT bit11)
           TBEN_L4_8IOL:O.Data[54].12   // IO-Link Port 4 - Output data word 4 (INT bit12)
           TBEN_L4_8IOL:O.Data[54].13   // IO-Link Port 4 - Output data word 4 (INT bit13)
           TBEN_L4_8IOL:O.Data[54].14   // IO-Link Port 4 - Output data word 4 (INT bit14)
           TBEN_L4_8IOL:O.Data[54].15   // IO-Link Port 4 - Output data word 4 (INT bit15)
           TBEN_L4_8IOL:O.Data[54].2   // IO-Link Port 4 - Output data word 4 (INT bit2)
           TBEN_L4_8IOL:O.Data[54].3   // IO-Link Port 4 - Output data word 4 (INT bit3)
           TBEN_L4_8IOL:O.Data[54].4   // IO-Link Port 4 - Output data word 4 (INT bit4)
           TBEN_L4_8IOL:O.Data[54].5   // IO-Link Port 4 - Output data word 4 (INT bit5)
           TBEN_L4_8IOL:O.Data[54].6   // IO-Link Port 4 - Output data word 4 (INT bit6)
           TBEN_L4_8IOL:O.Data[54].7   // IO-Link Port 4 - Output data word 4 (INT bit7)
           TBEN_L4_8IOL:O.Data[54].8   // IO-Link Port 4 - Output data word 4 (INT bit8)
           TBEN_L4_8IOL:O.Data[54].9   // IO-Link Port 4 - Output data word 4 (INT bit9)
           TBEN_L4_8IOL:O.Data[55]   // IO-Link Port 4 - Output data word 5
           TBEN_L4_8IOL:O.Data[55].0   // IO-Link Port 4 - Output data word 5 (INT bit0)
           TBEN_L4_8IOL:O.Data[55].1   // IO-Link Port 4 - Output data word 5 (INT bit1)
           TBEN_L4_8IOL:O.Data[55].10   // IO-Link Port 4 - Output data word 5 (INT bit10)
           TBEN_L4_8IOL:O.Data[55].11   // IO-Link Port 4 - Output data word 5 (INT bit11)
           TBEN_L4_8IOL:O.Data[55].12   // IO-Link Port 4 - Output data word 5 (INT bit12)
           TBEN_L4_8IOL:O.Data[55].13   // IO-Link Port 4 - Output data word 5 (INT bit13)
           TBEN_L4_8IOL:O.Data[55].14   // IO-Link Port 4 - Output data word 5 (INT bit14)
           TBEN_L4_8IOL:O.Data[55].15   // IO-Link Port 4 - Output data word 5 (INT bit15)
           TBEN_L4_8IOL:O.Data[55].2   // IO-Link Port 4 - Output data word 5 (INT bit2)
           TBEN_L4_8IOL:O.Data[55].3   // IO-Link Port 4 - Output data word 5 (INT bit3)
           TBEN_L4_8IOL:O.Data[55].4   // IO-Link Port 4 - Output data word 5 (INT bit4)
           TBEN_L4_8IOL:O.Data[55].5   // IO-Link Port 4 - Output data word 5 (INT bit5)
           TBEN_L4_8IOL:O.Data[55].6   // IO-Link Port 4 - Output data word 5 (INT bit6)
           TBEN_L4_8IOL:O.Data[55].7   // IO-Link Port 4 - Output data word 5 (INT bit7)
           TBEN_L4_8IOL:O.Data[55].8   // IO-Link Port 4 - Output data word 5 (INT bit8)
           TBEN_L4_8IOL:O.Data[55].9   // IO-Link Port 4 - Output data word 5 (INT bit9)
           TBEN_L4_8IOL:O.Data[56]   // IO-Link Port 4 - Output data word 6
           TBEN_L4_8IOL:O.Data[56].0   // IO-Link Port 4 - Output data word 6 (INT bit0)
           TBEN_L4_8IOL:O.Data[56].1   // IO-Link Port 4 - Output data word 6 (INT bit1)
           TBEN_L4_8IOL:O.Data[56].10   // IO-Link Port 4 - Output data word 6 (INT bit10)
           TBEN_L4_8IOL:O.Data[56].11   // IO-Link Port 4 - Output data word 6 (INT bit11)
           TBEN_L4_8IOL:O.Data[56].12   // IO-Link Port 4 - Output data word 6 (INT bit12)
           TBEN_L4_8IOL:O.Data[56].13   // IO-Link Port 4 - Output data word 6 (INT bit13)
           TBEN_L4_8IOL:O.Data[56].14   // IO-Link Port 4 - Output data word 6 (INT bit14)
           TBEN_L4_8IOL:O.Data[56].15   // IO-Link Port 4 - Output data word 6 (INT bit15)
           TBEN_L4_8IOL:O.Data[56].2   // IO-Link Port 4 - Output data word 6 (INT bit2)
           TBEN_L4_8IOL:O.Data[56].3   // IO-Link Port 4 - Output data word 6 (INT bit3)
           TBEN_L4_8IOL:O.Data[56].4   // IO-Link Port 4 - Output data word 6 (INT bit4)
           TBEN_L4_8IOL:O.Data[56].5   // IO-Link Port 4 - Output data word 6 (INT bit5)
           TBEN_L4_8IOL:O.Data[56].6   // IO-Link Port 4 - Output data word 6 (INT bit6)
           TBEN_L4_8IOL:O.Data[56].7   // IO-Link Port 4 - Output data word 6 (INT bit7)
           TBEN_L4_8IOL:O.Data[56].8   // IO-Link Port 4 - Output data word 6 (INT bit8)
           TBEN_L4_8IOL:O.Data[56].9   // IO-Link Port 4 - Output data word 6 (INT bit9)
           TBEN_L4_8IOL:O.Data[57]   // IO-Link Port 4 - Output data word 7
           TBEN_L4_8IOL:O.Data[57].0   // IO-Link Port 4 - Output data word 7 (INT bit0)
           TBEN_L4_8IOL:O.Data[57].1   // IO-Link Port 4 - Output data word 7 (INT bit1)
           TBEN_L4_8IOL:O.Data[57].10   // IO-Link Port 4 - Output data word 7 (INT bit10)
           TBEN_L4_8IOL:O.Data[57].11   // IO-Link Port 4 - Output data word 7 (INT bit11)
           TBEN_L4_8IOL:O.Data[57].12   // IO-Link Port 4 - Output data word 7 (INT bit12)
           TBEN_L4_8IOL:O.Data[57].13   // IO-Link Port 4 - Output data word 7 (INT bit13)
           TBEN_L4_8IOL:O.Data[57].14   // IO-Link Port 4 - Output data word 7 (INT bit14)
           TBEN_L4_8IOL:O.Data[57].15   // IO-Link Port 4 - Output data word 7 (INT bit15)
           TBEN_L4_8IOL:O.Data[57].2   // IO-Link Port 4 - Output data word 7 (INT bit2)
           TBEN_L4_8IOL:O.Data[57].3   // IO-Link Port 4 - Output data word 7 (INT bit3)
           TBEN_L4_8IOL:O.Data[57].4   // IO-Link Port 4 - Output data word 7 (INT bit4)
           TBEN_L4_8IOL:O.Data[57].5   // IO-Link Port 4 - Output data word 7 (INT bit5)
           TBEN_L4_8IOL:O.Data[57].6   // IO-Link Port 4 - Output data word 7 (INT bit6)
           TBEN_L4_8IOL:O.Data[57].7   // IO-Link Port 4 - Output data word 7 (INT bit7)
           TBEN_L4_8IOL:O.Data[57].8   // IO-Link Port 4 - Output data word 7 (INT bit8)
           TBEN_L4_8IOL:O.Data[57].9   // IO-Link Port 4 - Output data word 7 (INT bit9)
           TBEN_L4_8IOL:O.Data[58]   // IO-Link Port 4 - Output data word 8
           TBEN_L4_8IOL:O.Data[58].0   // IO-Link Port 4 - Output data word 8 (INT bit0)
           TBEN_L4_8IOL:O.Data[58].1   // IO-Link Port 4 - Output data word 8 (INT bit1)
           TBEN_L4_8IOL:O.Data[58].10   // IO-Link Port 4 - Output data word 8 (INT bit10)
           TBEN_L4_8IOL:O.Data[58].11   // IO-Link Port 4 - Output data word 8 (INT bit11)
           TBEN_L4_8IOL:O.Data[58].12   // IO-Link Port 4 - Output data word 8 (INT bit12)
           TBEN_L4_8IOL:O.Data[58].13   // IO-Link Port 4 - Output data word 8 (INT bit13)
           TBEN_L4_8IOL:O.Data[58].14   // IO-Link Port 4 - Output data word 8 (INT bit14)
           TBEN_L4_8IOL:O.Data[58].15   // IO-Link Port 4 - Output data word 8 (INT bit15)
           TBEN_L4_8IOL:O.Data[58].2   // IO-Link Port 4 - Output data word 8 (INT bit2)
           TBEN_L4_8IOL:O.Data[58].3   // IO-Link Port 4 - Output data word 8 (INT bit3)
           TBEN_L4_8IOL:O.Data[58].4   // IO-Link Port 4 - Output data word 8 (INT bit4)
           TBEN_L4_8IOL:O.Data[58].5   // IO-Link Port 4 - Output data word 8 (INT bit5)
           TBEN_L4_8IOL:O.Data[58].6   // IO-Link Port 4 - Output data word 8 (INT bit6)
           TBEN_L4_8IOL:O.Data[58].7   // IO-Link Port 4 - Output data word 8 (INT bit7)
           TBEN_L4_8IOL:O.Data[58].8   // IO-Link Port 4 - Output data word 8 (INT bit8)
           TBEN_L4_8IOL:O.Data[58].9   // IO-Link Port 4 - Output data word 8 (INT bit9)
           TBEN_L4_8IOL:O.Data[59]   // IO-Link Port 4 - Output data word 9
           TBEN_L4_8IOL:O.Data[59].0   // IO-Link Port 4 - Output data word 9 (INT bit0)
           TBEN_L4_8IOL:O.Data[59].1   // IO-Link Port 4 - Output data word 9 (INT bit1)
           TBEN_L4_8IOL:O.Data[59].10   // IO-Link Port 4 - Output data word 9 (INT bit10)
           TBEN_L4_8IOL:O.Data[59].11   // IO-Link Port 4 - Output data word 9 (INT bit11)
           TBEN_L4_8IOL:O.Data[59].12   // IO-Link Port 4 - Output data word 9 (INT bit12)
           TBEN_L4_8IOL:O.Data[59].13   // IO-Link Port 4 - Output data word 9 (INT bit13)
           TBEN_L4_8IOL:O.Data[59].14   // IO-Link Port 4 - Output data word 9 (INT bit14)
           TBEN_L4_8IOL:O.Data[59].15   // IO-Link Port 4 - Output data word 9 (INT bit15)
           TBEN_L4_8IOL:O.Data[59].2   // IO-Link Port 4 - Output data word 9 (INT bit2)
           TBEN_L4_8IOL:O.Data[59].3   // IO-Link Port 4 - Output data word 9 (INT bit3)
           TBEN_L4_8IOL:O.Data[59].4   // IO-Link Port 4 - Output data word 9 (INT bit4)
           TBEN_L4_8IOL:O.Data[59].5   // IO-Link Port 4 - Output data word 9 (INT bit5)
           TBEN_L4_8IOL:O.Data[59].6   // IO-Link Port 4 - Output data word 9 (INT bit6)
           TBEN_L4_8IOL:O.Data[59].7   // IO-Link Port 4 - Output data word 9 (INT bit7)
           TBEN_L4_8IOL:O.Data[59].8   // IO-Link Port 4 - Output data word 9 (INT bit8)
           TBEN_L4_8IOL:O.Data[59].9   // IO-Link Port 4 - Output data word 9 (INT bit9)
           TBEN_L4_8IOL:O.Data[5]   // IO-Link Port 1 - Output data word 3
           TBEN_L4_8IOL:O.Data[5].0   // IO-Link Port 1 - Output data word 3 (INT bit0)
           TBEN_L4_8IOL:O.Data[5].1   // IO-Link Port 1 - Output data word 3 (INT bit1)
           TBEN_L4_8IOL:O.Data[5].10   // IO-Link Port 1 - Output data word 3 (INT bit10)
           TBEN_L4_8IOL:O.Data[5].11   // IO-Link Port 1 - Output data word 3 (INT bit11)
           TBEN_L4_8IOL:O.Data[5].12   // IO-Link Port 1 - Output data word 3 (INT bit12)
           TBEN_L4_8IOL:O.Data[5].13   // IO-Link Port 1 - Output data word 3 (INT bit13)
           TBEN_L4_8IOL:O.Data[5].14   // IO-Link Port 1 - Output data word 3 (INT bit14)
           TBEN_L4_8IOL:O.Data[5].15   // IO-Link Port 1 - Output data word 3 (INT bit15)
           TBEN_L4_8IOL:O.Data[5].2   // IO-Link Port 1 - Output data word 3 (INT bit2)
           TBEN_L4_8IOL:O.Data[5].3   // IO-Link Port 1 - Output data word 3 (INT bit3)
           TBEN_L4_8IOL:O.Data[5].4   // IO-Link Port 1 - Output data word 3 (INT bit4)
           TBEN_L4_8IOL:O.Data[5].5   // IO-Link Port 1 - Output data word 3 (INT bit5)
           TBEN_L4_8IOL:O.Data[5].6   // IO-Link Port 1 - Output data word 3 (INT bit6)
           TBEN_L4_8IOL:O.Data[5].7   // IO-Link Port 1 - Output data word 3 (INT bit7)
           TBEN_L4_8IOL:O.Data[5].8   // IO-Link Port 1 - Output data word 3 (INT bit8)
           TBEN_L4_8IOL:O.Data[5].9   // IO-Link Port 1 - Output data word 3 (INT bit9)
           TBEN_L4_8IOL:O.Data[60]   // IO-Link Port 4 - Output data word 10
           TBEN_L4_8IOL:O.Data[60].0   // IO-Link Port 4 - Output data word 10 (INT bit0)
           TBEN_L4_8IOL:O.Data[60].1   // IO-Link Port 4 - Output data word 10 (INT bit1)
           TBEN_L4_8IOL:O.Data[60].10   // IO-Link Port 4 - Output data word 10 (INT bit10)
           TBEN_L4_8IOL:O.Data[60].11   // IO-Link Port 4 - Output data word 10 (INT bit11)
           TBEN_L4_8IOL:O.Data[60].12   // IO-Link Port 4 - Output data word 10 (INT bit12)
           TBEN_L4_8IOL:O.Data[60].13   // IO-Link Port 4 - Output data word 10 (INT bit13)
           TBEN_L4_8IOL:O.Data[60].14   // IO-Link Port 4 - Output data word 10 (INT bit14)
           TBEN_L4_8IOL:O.Data[60].15   // IO-Link Port 4 - Output data word 10 (INT bit15)
           TBEN_L4_8IOL:O.Data[60].2   // IO-Link Port 4 - Output data word 10 (INT bit2)
           TBEN_L4_8IOL:O.Data[60].3   // IO-Link Port 4 - Output data word 10 (INT bit3)
           TBEN_L4_8IOL:O.Data[60].4   // IO-Link Port 4 - Output data word 10 (INT bit4)
           TBEN_L4_8IOL:O.Data[60].5   // IO-Link Port 4 - Output data word 10 (INT bit5)
           TBEN_L4_8IOL:O.Data[60].6   // IO-Link Port 4 - Output data word 10 (INT bit6)
           TBEN_L4_8IOL:O.Data[60].7   // IO-Link Port 4 - Output data word 10 (INT bit7)
           TBEN_L4_8IOL:O.Data[60].8   // IO-Link Port 4 - Output data word 10 (INT bit8)
           TBEN_L4_8IOL:O.Data[60].9   // IO-Link Port 4 - Output data word 10 (INT bit9)
           TBEN_L4_8IOL:O.Data[61]   // IO-Link Port 4 - Output data word 11
           TBEN_L4_8IOL:O.Data[61].0   // IO-Link Port 4 - Output data word 11 (INT bit0)
           TBEN_L4_8IOL:O.Data[61].1   // IO-Link Port 4 - Output data word 11 (INT bit1)
           TBEN_L4_8IOL:O.Data[61].10   // IO-Link Port 4 - Output data word 11 (INT bit10)
           TBEN_L4_8IOL:O.Data[61].11   // IO-Link Port 4 - Output data word 11 (INT bit11)
           TBEN_L4_8IOL:O.Data[61].12   // IO-Link Port 4 - Output data word 11 (INT bit12)
           TBEN_L4_8IOL:O.Data[61].13   // IO-Link Port 4 - Output data word 11 (INT bit13)
           TBEN_L4_8IOL:O.Data[61].14   // IO-Link Port 4 - Output data word 11 (INT bit14)
           TBEN_L4_8IOL:O.Data[61].15   // IO-Link Port 4 - Output data word 11 (INT bit15)
           TBEN_L4_8IOL:O.Data[61].2   // IO-Link Port 4 - Output data word 11 (INT bit2)
           TBEN_L4_8IOL:O.Data[61].3   // IO-Link Port 4 - Output data word 11 (INT bit3)
           TBEN_L4_8IOL:O.Data[61].4   // IO-Link Port 4 - Output data word 11 (INT bit4)
           TBEN_L4_8IOL:O.Data[61].5   // IO-Link Port 4 - Output data word 11 (INT bit5)
           TBEN_L4_8IOL:O.Data[61].6   // IO-Link Port 4 - Output data word 11 (INT bit6)
           TBEN_L4_8IOL:O.Data[61].7   // IO-Link Port 4 - Output data word 11 (INT bit7)
           TBEN_L4_8IOL:O.Data[61].8   // IO-Link Port 4 - Output data word 11 (INT bit8)
           TBEN_L4_8IOL:O.Data[61].9   // IO-Link Port 4 - Output data word 11 (INT bit9)
           TBEN_L4_8IOL:O.Data[62]   // IO-Link Port 4 - Output data word 12
           TBEN_L4_8IOL:O.Data[62].0   // IO-Link Port 4 - Output data word 12 (INT bit0)
           TBEN_L4_8IOL:O.Data[62].1   // IO-Link Port 4 - Output data word 12 (INT bit1)
           TBEN_L4_8IOL:O.Data[62].10   // IO-Link Port 4 - Output data word 12 (INT bit10)
           TBEN_L4_8IOL:O.Data[62].11   // IO-Link Port 4 - Output data word 12 (INT bit11)
           TBEN_L4_8IOL:O.Data[62].12   // IO-Link Port 4 - Output data word 12 (INT bit12)
           TBEN_L4_8IOL:O.Data[62].13   // IO-Link Port 4 - Output data word 12 (INT bit13)
           TBEN_L4_8IOL:O.Data[62].14   // IO-Link Port 4 - Output data word 12 (INT bit14)
           TBEN_L4_8IOL:O.Data[62].15   // IO-Link Port 4 - Output data word 12 (INT bit15)
           TBEN_L4_8IOL:O.Data[62].2   // IO-Link Port 4 - Output data word 12 (INT bit2)
           TBEN_L4_8IOL:O.Data[62].3   // IO-Link Port 4 - Output data word 12 (INT bit3)
           TBEN_L4_8IOL:O.Data[62].4   // IO-Link Port 4 - Output data word 12 (INT bit4)
           TBEN_L4_8IOL:O.Data[62].5   // IO-Link Port 4 - Output data word 12 (INT bit5)
           TBEN_L4_8IOL:O.Data[62].6   // IO-Link Port 4 - Output data word 12 (INT bit6)
           TBEN_L4_8IOL:O.Data[62].7   // IO-Link Port 4 - Output data word 12 (INT bit7)
           TBEN_L4_8IOL:O.Data[62].8   // IO-Link Port 4 - Output data word 12 (INT bit8)
           TBEN_L4_8IOL:O.Data[62].9   // IO-Link Port 4 - Output data word 12 (INT bit9)
           TBEN_L4_8IOL:O.Data[63]   // IO-Link Port 4 - Output data word 13
